					(* Valuto la posizione attuale Y e la posizione di destinazione Y e l'ingombro massimo che posso avere durante il transito *)
					IF (Mission^.YPick - IngombroOttimizzatoY_InTransito/2 - OffsetSicurezza_Y <= WorkFootprint^[5].Y) OR //Posizione Pinza - Metà ingombro - Offset sicurezza <= Ingombro colonna 
						(Mission^.YPick + IngombroOttimizzatoY_InTransito/2 + OffsetSicurezza_Y >= WorkFootprint^[6].Y) THEN //Posizione Pinza - Metà ingombro - Offset sicurezza <= Ingombro colonna 
							Pinza_InIngombroColonne_Transito := TRUE;
					ELSE
							Pinza_InIngombroColonne_Transito := FALSE;
					END_IF
			END_CASE		
			(* Se sono in ingombro nella posizione attuale o nella posizione di destinazione, devo andare fuori-ingombro con la Y *)
			IF (Pinza_InIngombroColonne_Attuale OR Pinza_InIngombroColonne_Destinazione OR Pinza_InIngombroColonne_Transito) AND AreaInLavoroPositivaNegativa THEN 
				IF (AsseXInFinestraDiRiposo AND AsseYInFinestraDiRiposo AND AsseJInFinestraDiRiposo) THEN //Se sono in finestra di riposo con tutti gli assi non devo andare fuori-ingombro con la Y
					FuoriIngombroYNecessarioTMP := FALSE;
				ELSE
					FuoriIngombroYNecessarioTMP := TRUE;
				END_IF
			ELSE
				FuoriIngombroYNecessarioTMP := FALSE;
			END_IF
		END_IF
				
	WAMANAGER_CICLO_PRELIEVO_FALDA_VUOTI_END:
		CalcolaIngombro := TRUE;	
		
	WAMANAGER_CICLO_DEPOSITO_FALDA_VUOTI_RUN:
		IF CalcolaIngombro THEN
			CalcolaIngombro := FALSE;
			(* Definisco il tipo di area in cui si trova a lavorare il pallettizzatore *)
			AreaInLavoroPositiva := FALSE;
			AreaInLavoroNegativa := FALSE;
			AreaInLavoroPositivaNegativa := FALSE; 
			IF ModuleAx_X^.Ax^.AxRef^.NcToPlc.ActPos >= (WorkFootprint^[5].X + WorkFootprint^[5].XDim) AND 	//se la piazzola di prelievo ha quota maggiore rispetto le colonne centrali
				WorkArea^[Mission^.PPlace].X >= (WorkFootprint^[5].X + WorkFootprint^[5].XDim)  THEN //la piazzola di deposito è nella campata positiva
					AreaInLavoroPositiva := TRUE;
			ELSIF ModuleAx_X^.Ax^.AxRef^.NcToPlc.ActPos <= WorkFootprint^[5].X AND 	//se la piazzola di prelievo ha quota maggiore della piazzola di deposito e
				WorkArea^[Mission^.PPlace].X <= WorkFootprint^[5].X  THEN //la piazzola di deposito è nella campata negativa
					AreaInLavoroNegativa := TRUE;
			ELSE
				AreaInLavoroPositiva := FALSE;
				AreaInLavoroNegativa := FALSE;
				AreaInLavoroPositivaNegativa := TRUE;
			END_IF
			
			(**************************************************************************************************************************************************)
			(* Ingombro ottimizzato della pinza sul punto di prelievo *)
			(**************************************************************************************************************************************************)
			IngombroOttimizzatoX_InPuntoDiPrelievo := ABS(IngombroSuperficialePinzaMAX * SIN(deg_to_rad((ATAN(Larghezza/Lunghezza)*1/0.017+ Mission^.JPick))));
			IngombroOttimizzatoY_InPuntoDiPrelievo := ABS(IngombroSuperficialePinzaMAX * COS(deg_to_rad((ATAN(Larghezza/Lunghezza)*1/0.017+ Mission^.JPick))));
			(**************************************************************************************************************************************************)
			(* Ingombro ottimizzato della pinza sul punto di deposito *)
			(**************************************************************************************************************************************************)
			IngombroOttimizzatoX_InPuntoDiDeposito := ABS(IngombroSuperficialePinzaMAX * SIN(deg_to_rad((ATAN(Larghezza/Lunghezza)*1/0.017+ Mission^.JPlace))));
			IngombroOttimizzatoY_InPuntoDiDeposito := ABS(IngombroSuperficialePinzaMAX * COS(deg_to_rad((ATAN(Larghezza/Lunghezza)*1/0.017+ Mission^.JPlace))));
						
			(**************************************************************************************************************************************************)
			(**************************************************************************************************************************************************)
						
			(* Valuto la direzione della X *)
			DirezioneXPositiva := TFDirezioneAssePositiva(Posizione_Attuale:=ModuleAX_X^.Ax^.Status.ActPosition,Posizione_Finale:=Mission^.XPick);
			DirezioneXNegativa := NOT DirezioneXPositiva;
				
			(* Valuto se gli assi sono in finestra di prelievo *)
			AsseXInFinestraDiRiposo := TFAsseInFinestra(Posizione_Attuale:=ModuleAx_X^.Ax^.AxRef^.NcToPlc.ActPos,Posizione_Finale:=Mission^.XPick,FinestraDiControllo:=10);
			AsseYInFinestraDiRiposo := TFAsseInFinestra(Posizione_Attuale:=ModuleAx_Y^.Ax^.AxRef^.NcToPlc.ActPos,Posizione_Finale:=Mission^.YPick,FinestraDiControllo:=10);
			AsseJInFinestraDiRiposo := TFAsseInFinestra(Posizione_Attuale:=ModuleAx_J^.Ax^.AxRef^.NcToPlc.ActPos,Posizione_Finale:=Mission^.JPick,FinestraDiControllo:=5);
			(* Valuto se gli assi sono in finestra di destinazione *)
			AsseXInFinestraDiDestinazione := TFAsseInFinestra(Posizione_Attuale:=ModuleAx_X^.Ax^.AxRef^.NcToPlc.ActPos,Posizione_Finale:=Mission^.XPick,FinestraDiControllo:=10);
			AsseYInFinestraDiDestinazione := TFAsseInFinestra(Posizione_Attuale:=ModuleAx_Y^.Ax^.AxRef^.NcToPlc.ActPos,Posizione_Finale:=Mission^.YPick,FinestraDiControllo:=10);
			AsseJInFinestraDiDestinazione := TFAsseInFinestra(Posizione_Attuale:=ModuleAx_J^.Ax^.AxRef^.NcToPlc.ActPos,Posizione_Finale:=Mission^.JPick,FinestraDiControllo:=5);
			
			(**************************************************************************************************************************************************)
			(* Ingombro MASSIMO della pinza durante il transito *)
			(**************************************************************************************************************************************************)
			//Calcolo ingombro attuale
			IngombroOttimizzatoX_InTransito := ABS(IngombroSuperficialePinzaMAX * SIN(deg_to_rad((ATAN(Larghezza/Lunghezza)*1/0.017+ ModuleAx_J^.Ax^.AxRef^.NcToPlc.ActPos)))); //Ingombro Attuale direzione X
			IngombroOttimizzatoY_InTransito := ABS(IngombroSuperficialePinzaMAX * COS(deg_to_rad((ATAN(Larghezza/Lunghezza)*1/0.017+ ModuleAx_J^.Ax^.AxRef^.NcToPlc.ActPos)))); //Ingombro Attuale direzione Y		
			IF NOT AsseJInFinestraDiDestinazione THEN
				IF REAL_TO_INT(ModuleAx_J^.Ax^.AxRef^.NcToPlc.ActPos) <= REAL_TO_INT(Mission^.JPick) THEN
					FOR Angolo := REAL_TO_INT(ModuleAx_J^.Ax^.AxRef^.NcToPlc.ActPos) TO REAL_TO_INT(Mission^.JPick)  DO
						IF IngombroOttimizzatoX_InTransito < ABS(IngombroSuperficialePinzaMAX * SIN(deg_to_rad((ATAN(Larghezza/Lunghezza)*1/0.017+ Angolo)))) THEN
							IngombroOttimizzatoX_InTransito := ABS(IngombroSuperficialePinzaMAX * SIN(deg_to_rad((ATAN(Larghezza/Lunghezza)*1/0.017+ Angolo)))) ;
						END_IF
						IF IngombroOttimizzatoY_InTransito < ABS(IngombroSuperficialePinzaMAX * COS(deg_to_rad((ATAN(Larghezza/Lunghezza)*1/0.017+ Angolo)))) THEN
							IngombroOttimizzatoY_InTransito := ABS(IngombroSuperficialePinzaMAX * COS(deg_to_rad((ATAN(Larghezza/Lunghezza)*1/0.017+ Angolo))));
						END_IF
					END_FOR
				END_IF
			END_IF
		
			(* Valutazione colonne in base al verso del pallettizzatore *)
			CASE VERSO_PALLETTIZZATORE OF
				PALLETTIZZATORE_DX:	// Colonna 6:DX, 5:SX
					(* Valuto la posizione attuale *)
					IF (ModuleAX_Y^.Ax^.Status.ActPosition - IngombroY/2 - OffsetSicurezza_Y <= WorkFootprint^[6].Y) OR //Posizione Pinza - Metà ingombro - Offset sicurezza <= Ingombro colonna 
						(ModuleAX_Y^.Ax^.Status.ActPosition + IngombroY/2 + OffsetSicurezza_Y >= WorkFootprint^[5].Y) THEN //Posizione Pinza - Metà ingombro - Offset sicurezza <= Ingombro colonna 
							Pinza_InIngombroColonne_Attuale := TRUE;
					ELSE
							Pinza_InIngombroColonne_Attuale := FALSE;
					END_IF
					(* Valuto la posizione futura - Missione di prelievo *)
					IF (Mission^.YPick - IngombroOttimizzatoX_InPuntoDiPrelievo/2 - OffsetSicurezza_Y <= WorkFootprint^[6].Y) OR //Posizione Pinza - Metà ingombro - Offset sicurezza <= Ingombro colonna 
						(Mission^.YPick + IngombroOttimizzatoX_InPuntoDiPrelievo/2 + OffsetSicurezza_Y >= WorkFootprint^[5].Y) THEN //Posizione Pinza - Metà ingombro - Offset sicurezza <= Ingombro colonna 
							Pinza_InIngombroColonne_Destinazione := TRUE;
					ELSE
							Pinza_InIngombroColonne_Destinazione := FALSE;
					END_IF
					
					(* Valuto la posizione futura - Missione di Deposito *)
					IF (Mission^.YPick - IngombroOttimizzatoX_InPuntoDiDeposito/2 - OffsetSicurezza_Y <= WorkFootprint^[6].Y) OR //Posizione Pinza - Metà ingombro - Offset sicurezza <= Ingombro colonna 
						(Mission^.YPick + IngombroOttimizzatoX_InPuntoDiDeposito/2 + OffsetSicurezza_Y >= WorkFootprint^[5].Y) THEN //Posizione Pinza - Metà ingombro - Offset sicurezza <= Ingombro colonna 
							Pinza_InIngombroColonne_Destinazione := TRUE;
					ELSE
							Pinza_InIngombroColonne_Destinazione := FALSE;
					END_IF
					
					(* Valuto la posizione attuale Y e la posizione di destinazione Y e l'ingombro massimo che posso avere durante il transito *)
					IF (Mission^.YPick - IngombroOttimizzatoY_InTransito/2 - OffsetSicurezza_Y <= WorkFootprint^[6].Y) OR //Posizione Pinza - Metà ingombro - Offset sicurezza <= Ingombro colonna 
						(Mission^.YPick + IngombroOttimizzatoY_InTransito/2 + OffsetSicurezza_Y >= WorkFootprint^[5].Y) THEN //Posizione Pinza - Metà ingombro - Offset sicurezza <= Ingombro colonna 
							Pinza_InIngombroColonne_Transito := TRUE;
					ELSE
							Pinza_InIngombroColonne_Transito := FALSE;
					END_IF
						
				PALLETTIZZATORE_SX: // Colonna 6:SX, 5:DX
					(* Valuto la posizione attuale *)
					IF (ModuleAX_Y^.Ax^.Status.ActPosition - IngombroY/2 - OffsetSicurezza_Y <= WorkFootprint^[5].Y) OR //Posizione Pinza - Metà ingombro - Offset sicurezza <= Ingombro colonna 
						(ModuleAX_Y^.Ax^.Status.ActPosition + IngombroY/2 + OffsetSicurezza_Y >= WorkFootprint^[6].Y) THEN //Posizione Pinza - Metà ingombro - Offset sicurezza <= Ingombro colonna 
							Pinza_InIngombroColonne_Attuale := TRUE;
					ELSE
							Pinza_InIngombroColonne_Attuale := FALSE;
					END_IF
					(* Valuto la posizione futura - Missione di prelievo *)
					IF (Mission^.YPick - IngombroOttimizzatoX_InPuntoDiPrelievo/2 - OffsetSicurezza_Y <= WorkFootprint^[5].Y) OR //Posizione Pinza - Metà ingombro - Offset sicurezza <= Ingombro colonna 
						(Mission^.YPick + IngombroOttimizzatoX_InPuntoDiPrelievo/2 + OffsetSicurezza_Y >= WorkFootprint^[6].Y) THEN //Posizione Pinza - Metà ingombro - Offset sicurezza <= Ingombro colonna 
							Pinza_InIngombroColonne_Destinazione := TRUE;
					ELSE
							Pinza_InIngombroColonne_Destinazione := FALSE;
					END_IF
					
					(* Valuto la posizione futura - Missione di Deposito *)
					IF (Mission^.YPick - IngombroOttimizzatoX_InPuntoDiDeposito/2 - OffsetSicurezza_Y <= WorkFootprint^[5].Y) OR //Posizione Pinza - Metà ingombro - Offset sicurezza <= Ingombro colonna 
						(Mission^.YPick + IngombroOttimizzatoX_InPuntoDiDeposito/2 + OffsetSicurezza_Y >= WorkFootprint^[6].Y) THEN //Posizione Pinza - Metà ingombro - Offset sicurezza <= Ingombro colonna 
							Pinza_InIngombroColonne_Destinazione := TRUE;
					ELSE
							Pinza_InIngombroColonne_Destinazione := FALSE;
					END_IF
					
					(* Valuto la posizione attuale Y e la posizione di destinazione Y e l'ingombro massimo che posso avere durante il transito *)
					IF (Mission^.YPick - IngombroOttimizzatoY_InTransito/2 - OffsetSicurezza_Y <= WorkFootprint^[5].Y) OR //Posizione Pinza - Metà ingombro - Offset sicurezza <= Ingombro colonna 
						(Mission^.YPick + IngombroOttimizzatoY_InTransito/2 + OffsetSicurezza_Y >= WorkFootprint^[6].Y) THEN //Posizione Pinza - Metà ingombro - Offset sicurezza <= Ingombro colonna 
							Pinza_InIngombroColonne_Transito := TRUE;
					ELSE
							Pinza_InIngombroColonne_Transito := FALSE;
					END_IF
			END_CASE		
			(* Se sono in ingombro nella posizione attuale o nella posizione di destinazione, devo andare fuori-ingombro con la Y *)
			IF (Pinza_InIngombroColonne_Attuale OR Pinza_InIngombroColonne_Destinazione OR Pinza_InIngombroColonne_Transito) AND AreaInLavoroPositivaNegativa THEN 
				IF (AsseXInFinestraDiRiposo AND AsseYInFinestraDiRiposo AND AsseJInFinestraDiRiposo) THEN //Se sono in finestra di riposo con tutti gli assi non devo andare fuori-ingombro con la Y
					FuoriIngombroYNecessarioTMP := FALSE;
				ELSE
					FuoriIngombroYNecessarioTMP := TRUE;
				END_IF
			ELSE
				FuoriIngombroYNecessarioTMP := FALSE;
			END_IF
		END_IF
								
	WAMANAGER_CICLO_DEPOSITO_FALDA_VUOTI_END:
		CalcolaIngombro := TRUE;	
	
	WAMANAGER_CICLO_FALDA_INIT:
		CalcolaIngombro := TRUE;	
	
	WAMANAGER_CICLO_PRELIEVO_FALDA_RUN:
		IF CalcolaIngombro THEN
			CalcolaIngombro := FALSE;
			(* Definisco il tipo di area in cui si trova a lavorare il pallettizzatore *)
			AreaInLavoroPositiva := FALSE;
			AreaInLavoroNegativa := FALSE;
			AreaInLavoroPositivaNegativa := TRUE; 
			
			(**************************************************************************************************************************************************)
			(* Ingombro ottimizzato della pinza sul punto di prelievo *)
			(**************************************************************************************************************************************************)
			IngombroOttimizzatoX_InPuntoDiPrelievo := ABS(IngombroSuperficialePinzaMAX * SIN(deg_to_rad((ATAN(Larghezza/Lunghezza)*1/0.017+ Mission^.JPick))));
			IngombroOttimizzatoY_InPuntoDiPrelievo := ABS(IngombroSuperficialePinzaMAX * COS(deg_to_rad((ATAN(Larghezza/Lunghezza)*1/0.017+ Mission^.JPick))));
			(**************************************************************************************************************************************************)
			(* Ingombro ottimizzato della pinza sul punto di deposito *)
			(**************************************************************************************************************************************************)
			IngombroOttimizzatoX_InPuntoDiDeposito := ABS(IngombroSuperficialePinzaMAX * SIN(deg_to_rad((ATAN(Larghezza/Lunghezza)*1/0.017+ Mission^.JPlace))));
			IngombroOttimizzatoY_InPuntoDiDeposito := ABS(IngombroSuperficialePinzaMAX * COS(deg_to_rad((ATAN(Larghezza/Lunghezza)*1/0.017+ Mission^.JPlace))));
						
			(**************************************************************************************************************************************************)
			(**************************************************************************************************************************************************)
						
			(* Valuto la direzione della X *)
			DirezioneXPositiva := TFDirezioneAssePositiva(Posizione_Attuale:=ModuleAX_X^.Ax^.Status.ActPosition,Posizione_Finale:=Mission^.XPick);
			DirezioneXNegativa := NOT DirezioneXPositiva;
				
			(* Valuto se gli assi sono in finestra di prelievo *)
			AsseXInFinestraDiRiposo := TFAsseInFinestra(Posizione_Attuale:=ModuleAx_X^.Ax^.AxRef^.NcToPlc.ActPos,Posizione_Finale:=Mission^.XPick,FinestraDiControllo:=10);
			AsseYInFinestraDiRiposo := TFAsseInFinestra(Posizione_Attuale:=ModuleAx_Y^.Ax^.AxRef^.NcToPlc.ActPos,Posizione_Finale:=Mission^.YPick,FinestraDiControllo:=10);
			AsseJInFinestraDiRiposo := TFAsseInFinestra(Posizione_Attuale:=ModuleAx_J^.Ax^.AxRef^.NcToPlc.ActPos,Posizione_Finale:=Mission^.JPick,FinestraDiControllo:=5);
			(* Valuto se gli assi sono in finestra di destinazione *)
			AsseXInFinestraDiDestinazione := TFAsseInFinestra(Posizione_Attuale:=ModuleAx_X^.Ax^.AxRef^.NcToPlc.ActPos,Posizione_Finale:=Mission^.XPick,FinestraDiControllo:=10);
			AsseYInFinestraDiDestinazione := TFAsseInFinestra(Posizione_Attuale:=ModuleAx_Y^.Ax^.AxRef^.NcToPlc.ActPos,Posizione_Finale:=Mission^.YPick,FinestraDiControllo:=10);
			AsseJInFinestraDiDestinazione := TFAsseInFinestra(Posizione_Attuale:=ModuleAx_J^.Ax^.AxRef^.NcToPlc.ActPos,Posizione_Finale:=Mission^.JPick,FinestraDiControllo:=5);
			
			(**************************************************************************************************************************************************)
			(* Ingombro MASSIMO della pinza durante il transito *)
			(**************************************************************************************************************************************************)
			//Calcolo ingombro attuale
			IngombroOttimizzatoX_InTransito := ABS(IngombroSuperficialePinzaMAX * SIN(deg_to_rad((ATAN(Larghezza/Lunghezza)*1/0.017+ ModuleAx_J^.Ax^.AxRef^.NcToPlc.ActPos)))); //Ingombro Attuale direzione X
			IngombroOttimizzatoY_InTransito := ABS(IngombroSuperficialePinzaMAX * COS(deg_to_rad((ATAN(Larghezza/Lunghezza)*1/0.017+ ModuleAx_J^.Ax^.AxRef^.NcToPlc.ActPos)))); //Ingombro Attuale direzione Y		
			IF NOT AsseJInFinestraDiDestinazione THEN
				IF REAL_TO_INT(ModuleAx_J^.Ax^.AxRef^.NcToPlc.ActPos) <= REAL_TO_INT(Mission^.JPick) THEN
					FOR Angolo := REAL_TO_INT(ModuleAx_J^.Ax^.AxRef^.NcToPlc.ActPos) TO REAL_TO_INT(Mission^.JPick)  DO
						IF IngombroOttimizzatoX_InTransito < ABS(IngombroSuperficialePinzaMAX * SIN(deg_to_rad((ATAN(Larghezza/Lunghezza)*1/0.017+ Angolo)))) THEN
							IngombroOttimizzatoX_InTransito := ABS(IngombroSuperficialePinzaMAX * SIN(deg_to_rad((ATAN(Larghezza/Lunghezza)*1/0.017+ Angolo)))) ;
						END_IF
						IF IngombroOttimizzatoY_InTransito < ABS(IngombroSuperficialePinzaMAX * COS(deg_to_rad((ATAN(Larghezza/Lunghezza)*1/0.017+ Angolo)))) THEN
							IngombroOttimizzatoY_InTransito := ABS(IngombroSuperficialePinzaMAX * COS(deg_to_rad((ATAN(Larghezza/Lunghezza)*1/0.017+ Angolo))));
						END_IF
					END_FOR
				END_IF
			END_IF
		
			(* Valutazione colonne in base al verso del pallettizzatore *)
			CASE VERSO_PALLETTIZZATORE OF
				PALLETTIZZATORE_DX:	// Colonna 6:DX, 5:SX
					(* Valuto la posizione attuale *)
					IF (ModuleAX_Y^.Ax^.Status.ActPosition - IngombroY/2 - OffsetSicurezza_Y <= WorkFootprint^[6].Y) OR //Posizione Pinza - Metà ingombro - Offset sicurezza <= Ingombro colonna 
						(ModuleAX_Y^.Ax^.Status.ActPosition + IngombroY/2 + OffsetSicurezza_Y >= WorkFootprint^[5].Y) THEN //Posizione Pinza - Metà ingombro - Offset sicurezza <= Ingombro colonna 
							Pinza_InIngombroColonne_Attuale := TRUE;
					ELSE
							Pinza_InIngombroColonne_Attuale := FALSE;
					END_IF
					(* Valuto la posizione futura - Missione di prelievo *)
					IF (Mission^.YPick - IngombroOttimizzatoX_InPuntoDiPrelievo/2 - OffsetSicurezza_Y <= WorkFootprint^[6].Y) OR //Posizione Pinza - Metà ingombro - Offset sicurezza <= Ingombro colonna 
						(Mission^.YPick + IngombroOttimizzatoX_InPuntoDiPrelievo/2 + OffsetSicurezza_Y >= WorkFootprint^[5].Y) THEN //Posizione Pinza - Metà ingombro - Offset sicurezza <= Ingombro colonna 
							Pinza_InIngombroColonne_Destinazione := TRUE;
					ELSE
							Pinza_InIngombroColonne_Destinazione := FALSE;
					END_IF
					
					(* Valuto la posizione futura - Missione di Deposito *)
					IF (Mission^.YPick - IngombroOttimizzatoX_InPuntoDiDeposito/2 - OffsetSicurezza_Y <= WorkFootprint^[6].Y) OR //Posizione Pinza - Metà ingombro - Offset sicurezza <= Ingombro colonna 
						(Mission^.YPick + IngombroOttimizzatoX_InPuntoDiDeposito/2 + OffsetSicurezza_Y >= WorkFootprint^[5].Y) THEN //Posizione Pinza - Metà ingombro - Offset sicurezza <= Ingombro colonna 
							Pinza_InIngombroColonne_Destinazione := TRUE;
					ELSE
							Pinza_InIngombroColonne_Destinazione := FALSE;
					END_IF
					
					(* Valuto la posizione attuale Y e la posizione di destinazione Y e l'ingombro massimo che posso avere durante il transito *)
					IF (Mission^.YPick - IngombroOttimizzatoY_InTransito/2 - OffsetSicurezza_Y <= WorkFootprint^[6].Y) OR //Posizione Pinza - Metà ingombro - Offset sicurezza <= Ingombro colonna 
						(Mission^.YPick + IngombroOttimizzatoY_InTransito/2 + OffsetSicurezza_Y >= WorkFootprint^[5].Y) THEN //Posizione Pinza - Metà ingombro - Offset sicurezza <= Ingombro colonna 
							Pinza_InIngombroColonne_Transito := TRUE;
					ELSE
							Pinza_InIngombroColonne_Transito := FALSE;
					END_IF
						
				PALLETTIZZATORE_SX: // Colonna 6:SX, 5:DX
					(* Valuto la posizione attuale *)
					IF (ModuleAX_Y^.Ax^.Status.ActPosition - IngombroY/2 - OffsetSicurezza_Y <= WorkFootprint^[5].Y) OR //Posizione Pinza - Metà ingombro - Offset sicurezza <= Ingombro colonna 
						(ModuleAX_Y^.Ax^.Status.ActPosition + IngombroY/2 + OffsetSicurezza_Y >= WorkFootprint^[6].Y) THEN //Posizione Pinza - Metà ingombro - Offset sicurezza <= Ingombro colonna 
							Pinza_InIngombroColonne_Attuale := TRUE;
					ELSE
							Pinza_InIngombroColonne_Attuale := FALSE;
					END_IF
					(* Valuto la posizione futura - Missione di prelievo *)
					IF (Mission^.YPick - IngombroOttimizzatoX_InPuntoDiPrelievo/2 - OffsetSicurezza_Y <= WorkFootprint^[5].Y) OR //Posizione Pinza - Metà ingombro - Offset sicurezza <= Ingombro colonna 
						(Mission^.YPick + IngombroOttimizzatoX_InPuntoDiPrelievo/2 + OffsetSicurezza_Y >= WorkFootprint^[6].Y) THEN //Posizione Pinza - Metà ingombro - Offset sicurezza <= Ingombro colonna 
							Pinza_InIngombroColonne_Destinazione := TRUE;
					ELSE
							Pinza_InIngombroColonne_Destinazione := FALSE;
					END_IF
					
					(* Valuto la posizione futura - Missione di Deposito *)
					IF (Mission^.YPick - IngombroOttimizzatoX_InPuntoDiDeposito/2 - OffsetSicurezza_Y <= WorkFootprint^[5].Y) OR //Posizione Pinza - Metà ingombro - Offset sicurezza <= Ingombro colonna 
						(Mission^.YPick + IngombroOttimizzatoX_InPuntoDiDeposito/2 + OffsetSicurezza_Y >= WorkFootprint^[6].Y) THEN //Posizione Pinza - Metà ingombro - Offset sicurezza <= Ingombro colonna 
							Pinza_InIngombroColonne_Destinazione := TRUE;
					ELSE
							Pinza_InIngombroColonne_Destinazione := FALSE;
					END_IF
					
					(* Valuto la posizione attuale Y e la posizione di destinazione Y e l'ingombro massimo che posso avere durante il transito *)
					IF (Mission^.YPick - IngombroOttimizzatoY_InTransito/2 - OffsetSicurezza_Y <= WorkFootprint^[5].Y) OR //Posizione Pinza - Metà ingombro - Offset sicurezza <= Ingombro colonna 
						(Mission^.YPick + IngombroOttimizzatoY_InTransito/2 + OffsetSicurezza_Y >= WorkFootprint^[6].Y) THEN //Posizione Pinza - Metà ingombro - Offset sicurezza <= Ingombro colonna 
							Pinza_InIngombroColonne_Transito := TRUE;
					ELSE
							Pinza_InIngombroColonne_Transito := FALSE;
					END_IF
			END_CASE		
			(* Se sono in ingombro nella posizione attuale o nella posizione di destinazione, devo andare fuori-ingombro con la Y *)
			IF (Pinza_InIngombroColonne_Attuale OR Pinza_InIngombroColonne_Destinazione OR Pinza_InIngombroColonne_Transito) THEN 
				IF (AsseXInFinestraDiRiposo AND AsseYInFinestraDiRiposo AND AsseJInFinestraDiRiposo) THEN //Se sono in finestra di riposo con tutti gli assi non devo andare fuori-ingombro con la Y
					FuoriIngombroYNecessarioTMP := FALSE;
				ELSE
					FuoriIngombroYNecessarioTMP := TRUE;
				END_IF
			ELSE
				FuoriIngombroYNecessarioTMP := FALSE;
			END_IF
		END_IF		
																
	WAMANAGER_CICLO_PRELIEVO_FALDA_END:
		CalcolaIngombro := TRUE;	
			
	WAMANAGER_CICLO_DEPOSITO_FALDA_RUN:
		IF CalcolaIngombro THEN
			CalcolaIngombro := FALSE;
			(* Definisco il tipo di area in cui si trova a lavorare il pallettizzatore *)
			AreaInLavoroPositiva := FALSE;
			AreaInLavoroNegativa := FALSE;
			AreaInLavoroPositivaNegativa := TRUE; 
			
			IF ModuleAx_X^.Ax^.AxRef^.NcToPlc.ActPos >= (WorkFootprint^[5].X + WorkFootprint^[5].XDim) AND 	//se la piazzola di prelievo ha quota maggiore rispetto le colonne centrali
				WorkArea^[Mission^.PPlace].X >= (WorkFootprint^[5].X + WorkFootprint^[5].XDim)  THEN //la piazzola di deposito è nella campata positiva
					AreaInLavoroPositiva := TRUE;
			ELSIF ModuleAx_X^.Ax^.AxRef^.NcToPlc.ActPos <= WorkFootprint^[5].X AND 	//se la piazzola di prelievo ha quota maggiore della piazzola di deposito e
				WorkArea^[Mission^.PPlace].X <= WorkFootprint^[5].X  THEN //la piazzola di deposito è nella campata negativa
					AreaInLavoroNegativa := TRUE;
			ELSE
				AreaInLavoroPositiva := FALSE;
				AreaInLavoroNegativa := FALSE;
				AreaInLavoroPositivaNegativa := TRUE;
			END_IF
			
			(**************************************************************************************************************************************************)
			(* Ingombro ottimizzato della pinza sul punto di prelievo *)
			(**************************************************************************************************************************************************)
			IngombroOttimizzatoX_InPuntoDiPrelievo := ABS(IngombroSuperficialePinzaMAX * SIN(deg_to_rad((ATAN(Larghezza/Lunghezza)*1/0.017+ Mission^.JPick))));
			IngombroOttimizzatoY_InPuntoDiPrelievo := ABS(IngombroSuperficialePinzaMAX * COS(deg_to_rad((ATAN(Larghezza/Lunghezza)*1/0.017+ Mission^.JPick))));
			(**************************************************************************************************************************************************)
			(* Ingombro ottimizzato della pinza sul punto di deposito *)
			(**************************************************************************************************************************************************)
			IngombroOttimizzatoX_InPuntoDiDeposito := ABS(IngombroSuperficialePinzaMAX * SIN(deg_to_rad((ATAN(Larghezza/Lunghezza)*1/0.017+ Mission^.JPlace))));
			IngombroOttimizzatoY_InPuntoDiDeposito := ABS(IngombroSuperficialePinzaMAX * COS(deg_to_rad((ATAN(Larghezza/Lunghezza)*1/0.017+ Mission^.JPlace))));
						
			(**************************************************************************************************************************************************)
			(**************************************************************************************************************************************************)
						
			(* Valuto la direzione della X *)
			DirezioneXPositiva := TFDirezioneAssePositiva(Posizione_Attuale:=ModuleAX_X^.Ax^.Status.ActPosition,Posizione_Finale:=Mission^.XPick);
			DirezioneXNegativa := NOT DirezioneXPositiva;
				
			(* Valuto se gli assi sono in finestra di prelievo *)
			AsseXInFinestraDiRiposo := TFAsseInFinestra(Posizione_Attuale:=ModuleAx_X^.Ax^.AxRef^.NcToPlc.ActPos,Posizione_Finale:=Mission^.XPick,FinestraDiControllo:=10);
			AsseYInFinestraDiRiposo := TFAsseInFinestra(Posizione_Attuale:=ModuleAx_Y^.Ax^.AxRef^.NcToPlc.ActPos,Posizione_Finale:=Mission^.YPick,FinestraDiControllo:=10);
			AsseJInFinestraDiRiposo := TFAsseInFinestra(Posizione_Attuale:=ModuleAx_J^.Ax^.AxRef^.NcToPlc.ActPos,Posizione_Finale:=Mission^.JPick,FinestraDiControllo:=5);
			(* Valuto se gli assi sono in finestra di destinazione *)
			AsseXInFinestraDiDestinazione := TFAsseInFinestra(Posizione_Attuale:=ModuleAx_X^.Ax^.AxRef^.NcToPlc.ActPos,Posizione_Finale:=Mission^.XPick,FinestraDiControllo:=10);
			AsseYInFinestraDiDestinazione := TFAsseInFinestra(Posizione_Attuale:=ModuleAx_Y^.Ax^.AxRef^.NcToPlc.ActPos,Posizione_Finale:=Mission^.YPick,FinestraDiControllo:=10);
			AsseJInFinestraDiDestinazione := TFAsseInFinestra(Posizione_Attuale:=ModuleAx_J^.Ax^.AxRef^.NcToPlc.ActPos,Posizione_Finale:=Mission^.JPick,FinestraDiControllo:=5);
			
			(**************************************************************************************************************************************************)
			(* Ingombro MASSIMO della pinza durante il transito *)
			(**************************************************************************************************************************************************)
			//Calcolo ingombro attuale
			IngombroOttimizzatoX_InTransito := ABS(IngombroSuperficialePinzaMAX * SIN(deg_to_rad((ATAN(Larghezza/Lunghezza)*1/0.017+ ModuleAx_J^.Ax^.AxRef^.NcToPlc.ActPos)))); //Ingombro Attuale direzione X
			IngombroOttimizzatoY_InTransito := ABS(IngombroSuperficialePinzaMAX * COS(deg_to_rad((ATAN(Larghezza/Lunghezza)*1/0.017+ ModuleAx_J^.Ax^.AxRef^.NcToPlc.ActPos)))); //Ingombro Attuale direzione Y		
			IF NOT AsseJInFinestraDiDestinazione THEN
				IF REAL_TO_INT(ModuleAx_J^.Ax^.AxRef^.NcToPlc.ActPos) <= REAL_TO_INT(Mission^.JPick) THEN
					FOR Angolo := REAL_TO_INT(ModuleAx_J^.Ax^.AxRef^.NcToPlc.ActPos) TO REAL_TO_INT(Mission^.JPick)  DO
						IF IngombroOttimizzatoX_InTransito < ABS(IngombroSuperficialePinzaMAX * SIN(deg_to_rad((ATAN(Larghezza/Lunghezza)*1/0.017+ Angolo)))) THEN
							IngombroOttimizzatoX_InTransito := ABS(IngombroSuperficialePinzaMAX * SIN(deg_to_rad((ATAN(Larghezza/Lunghezza)*1/0.017+ Angolo)))) ;
						END_IF
						IF IngombroOttimizzatoY_InTransito < ABS(IngombroSuperficialePinzaMAX * COS(deg_to_rad((ATAN(Larghezza/Lunghezza)*1/0.017+ Angolo)))) THEN
							IngombroOttimizzatoY_InTransito := ABS(IngombroSuperficialePinzaMAX * COS(deg_to_rad((ATAN(Larghezza/Lunghezza)*1/0.017+ Angolo))));
						END_IF
					END_FOR
				END_IF
			END_IF
		
			(* Valutazione colonne in base al verso del pallettizzatore *)
			CASE VERSO_PALLETTIZZATORE OF
				PALLETTIZZATORE_DX:	// Colonna 6:DX, 5:SX
					(* Valuto la posizione attuale *)
					IF (ModuleAX_Y^.Ax^.Status.ActPosition - IngombroY/2 - OffsetSicurezza_Y <= WorkFootprint^[6].Y) OR //Posizione Pinza - Metà ingombro - Offset sicurezza <= Ingombro colonna 
						(ModuleAX_Y^.Ax^.Status.ActPosition + IngombroY/2 + OffsetSicurezza_Y >= WorkFootprint^[5].Y) THEN //Posizione Pinza - Metà ingombro - Offset sicurezza <= Ingombro colonna 
							Pinza_InIngombroColonne_Attuale := TRUE;
					ELSE
							Pinza_InIngombroColonne_Attuale := FALSE;
					END_IF
					(* Valuto la posizione futura - Missione di prelievo *)
					IF (Mission^.YPick - IngombroOttimizzatoX_InPuntoDiPrelievo/2 - OffsetSicurezza_Y <= WorkFootprint^[6].Y) OR //Posizione Pinza - Metà ingombro - Offset sicurezza <= Ingombro colonna 
						(Mission^.YPick + IngombroOttimizzatoX_InPuntoDiPrelievo/2 + OffsetSicurezza_Y >= WorkFootprint^[5].Y) THEN //Posizione Pinza - Metà ingombro - Offset sicurezza <= Ingombro colonna 
							Pinza_InIngombroColonne_Destinazione := TRUE;
					ELSE
							Pinza_InIngombroColonne_Destinazione := FALSE;
					END_IF
					
					(* Valuto la posizione futura - Missione di Deposito *)
					IF (Mission^.YPick - IngombroOttimizzatoX_InPuntoDiDeposito/2 - OffsetSicurezza_Y <= WorkFootprint^[6].Y) OR //Posizione Pinza - Metà ingombro - Offset sicurezza <= Ingombro colonna 
						(Mission^.YPick + IngombroOttimizzatoX_InPuntoDiDeposito/2 + OffsetSicurezza_Y >= WorkFootprint^[5].Y) THEN //Posizione Pinza - Metà ingombro - Offset sicurezza <= Ingombro colonna 
							Pinza_InIngombroColonne_Destinazione := TRUE;
					ELSE
							Pinza_InIngombroColonne_Destinazione := FALSE;
					END_IF
					
					(* Valuto la posizione attuale Y e la posizione di destinazione Y e l'ingombro massimo che posso avere durante il transito *)
					IF (Mission^.YPick - IngombroOttimizzatoY_InTransito/2 - OffsetSicurezza_Y <= WorkFootprint^[6].Y) OR //Posizione Pinza - Metà ingombro - Offset sicurezza <= Ingombro colonna 
						(Mission^.YPick + IngombroOttimizzatoY_InTransito/2 + OffsetSicurezza_Y >= WorkFootprint^[5].Y) THEN //Posizione Pinza - Metà ingombro - Offset sicurezza <= Ingombro colonna 
							Pinza_InIngombroColonne_Transito := TRUE;
					ELSE
							Pinza_InIngombroColonne_Transito := FALSE;
					END_IF
						
				PALLETTIZZATORE_SX: // Colonna 6:SX, 5:DX
					(* Valuto la posizione attuale *)
					IF (ModuleAX_Y^.Ax^.Status.ActPosition - IngombroY/2 - OffsetSicurezza_Y <= WorkFootprint^[5].Y) OR //Posizione Pinza - Metà ingombro - Offset sicurezza <= Ingombro colonna 
						(ModuleAX_Y^.Ax^.Status.ActPosition + IngombroY/2 + OffsetSicurezza_Y >= WorkFootprint^[6].Y) THEN //Posizione Pinza - Metà ingombro - Offset sicurezza <= Ingombro colonna 
							Pinza_InIngombroColonne_Attuale := TRUE;
					ELSE
							Pinza_InIngombroColonne_Attuale := FALSE;
					END_IF
					(* Valuto la posizione futura - Missione di prelievo *)
					IF (Mission^.YPick - IngombroOttimizzatoX_InPuntoDiPrelievo/2 - OffsetSicurezza_Y <= WorkFootprint^[5].Y) OR //Posizione Pinza - Metà ingombro - Offset sicurezza <= Ingombro colonna 
						(Mission^.YPick + IngombroOttimizzatoX_InPuntoDiPrelievo/2 + OffsetSicurezza_Y >= WorkFootprint^[6].Y) THEN //Posizione Pinza - Metà ingombro - Offset sicurezza <= Ingombro colonna 
							Pinza_InIngombroColonne_Destinazione := TRUE;
					ELSE
							Pinza_InIngombroColonne_Destinazione := FALSE;
					END_IF
					
					(* Valuto la posizione futura - Missione di Deposito *)
					IF (Mission^.YPick - IngombroOttimizzatoX_InPuntoDiDeposito/2 - OffsetSicurezza_Y <= WorkFootprint^[5].Y) OR //Posizione Pinza - Metà ingombro - Offset sicurezza <= Ingombro colonna 
						(Mission^.YPick + IngombroOttimizzatoX_InPuntoDiDeposito/2 + OffsetSicurezza_Y >= WorkFootprint^[6].Y) THEN //Posizione Pinza - Metà ingombro - Offset sicurezza <= Ingombro colonna 
							Pinza_InIngombroColonne_Destinazione := TRUE;
					ELSE
							Pinza_InIngombroColonne_Destinazione := FALSE;
					END_IF
					
					(* Valuto la posizione attuale Y e la posizione di destinazione Y e l'ingombro massimo che posso avere durante il transito *)
					IF (Mission^.YPick - IngombroOttimizzatoY_InTransito/2 - OffsetSicurezza_Y <= WorkFootprint^[5].Y) OR //Posizione Pinza - Metà ingombro - Offset sicurezza <= Ingombro colonna 
						(Mission^.YPick + IngombroOttimizzatoY_InTransito/2 + OffsetSicurezza_Y >= WorkFootprint^[6].Y) THEN //Posizione Pinza - Metà ingombro - Offset sicurezza <= Ingombro colonna 
							Pinza_InIngombroColonne_Transito := TRUE;
					ELSE
							Pinza_InIngombroColonne_Transito := FALSE;
					END_IF
			END_CASE		
			(* Se sono in ingombro nella posizione attuale o nella posizione di destinazione, devo andare fuori-ingombro con la Y *)
			IF (Pinza_InIngombroColonne_Attuale OR Pinza_InIngombroColonne_Destinazione OR Pinza_InIngombroColonne_Transito) THEN 
				IF (AsseXInFinestraDiRiposo AND AsseYInFinestraDiRiposo AND AsseJInFinestraDiRiposo) THEN //Se sono in finestra di riposo con tutti gli assi non devo andare fuori-ingombro con la Y
					FuoriIngombroYNecessarioTMP := FALSE;
				ELSE
					FuoriIngombroYNecessarioTMP := TRUE;
				END_IF
			ELSE
				FuoriIngombroYNecessarioTMP := FALSE;
			END_IF
		END_IF
			
	WAMANAGER_CICLO_DEPOSITO_FALDA_END:
		CalcolaIngombro := TRUE;	

	WAMANAGER_CICLO_PACCO_INIT:
		CalcolaIngombro := TRUE;	
	
	WAMANAGER_CICLO_PRELIEVO_PACCO_RUN:
		
		IF CalcolaIngombro THEN
			CalcolaIngombro := FALSE;
			(* Definisco il tipo di area in cui si trova a lavorare il pallettizzatore *)
			AreaInLavoroPositiva := FALSE;
			AreaInLavoroNegativa := FALSE;
			AreaInLavoroPositivaNegativa := TRUE; 
			CASE Mission^.JPickVO OF
				(* Verticale *)
				0:	
					IF ModuleAx_X^.Ax^.AxRef^.NcToPlc.ActPos <= WorkFootprint^[5].X AND 
						WorkPickPoint^[Mission^.PPick].Xv <= WorkFootprint^[5].X THEN
							AreaInLavoroNegativa := TRUE;
					ELSIF ModuleAx_X^.Ax^.AxRef^.NcToPlc.ActPos >= WorkFootprint^[5].X AND 
						WorkPickPoint^[Mission^.PPick].Xv >= WorkFootprint^[5].X THEN
							AreaInLavoroPositiva := TRUE;
					ELSE
						AreaInLavoroPositiva := FALSE;
						AreaInLavoroNegativa := FALSE;
						AreaInLavoroPositivaNegativa := TRUE;
					END_IF
					
				(* Orrizontale *)
				1: 
					IF ModuleAx_X^.Ax^.AxRef^.NcToPlc.ActPos <= WorkFootprint^[5].X AND 
						WorkPickPoint^[Mission^.PPick].Xh <= WorkFootprint^[5].X THEN
							AreaInLavoroNegativa := TRUE;
					ELSIF ModuleAx_X^.Ax^.AxRef^.NcToPlc.ActPos >= (WorkFootprint^[5].X + WorkFootprint^[5].XDim) AND 
						WorkPickPoint^[Mission^.PPick].Xh >= (WorkFootprint^[5].X + WorkFootprint^[5].XDim) THEN
							AreaInLavoroPositiva := TRUE;
					ELSE
						AreaInLavoroPositiva := FALSE;
						AreaInLavoroNegativa := FALSE;
						AreaInLavoroPositivaNegativa := TRUE;
					END_IF
			END_CASE
			
			(**************************************************************************************************************************************************)
			(* Ingombro ottimizzato della pinza sul punto di prelievo *)
			(**************************************************************************************************************************************************)
			IngombroOttimizzatoX_InPuntoDiPrelievo := ABS(IngombroSuperficialePinzaMAX * SIN(deg_to_rad((ATAN(Larghezza/Lunghezza)*1/0.017+ Mission^.JPick))));
			IngombroOttimizzatoY_InPuntoDiPrelievo := ABS(IngombroSuperficialePinzaMAX * COS(deg_to_rad((ATAN(Larghezza/Lunghezza)*1/0.017+ Mission^.JPick))));
			(**************************************************************************************************************************************************)
			(* Ingombro ottimizzato della pinza sul punto di deposito *)
			(**************************************************************************************************************************************************)
			IngombroOttimizzatoX_InPuntoDiDeposito := ABS(IngombroSuperficialePinzaMAX * SIN(deg_to_rad((ATAN(Larghezza/Lunghezza)*1/0.017+ Mission^.JPlace))));
			IngombroOttimizzatoY_InPuntoDiDeposito := ABS(IngombroSuperficialePinzaMAX * COS(deg_to_rad((ATAN(Larghezza/Lunghezza)*1/0.017+ Mission^.JPlace))));
						
			(**************************************************************************************************************************************************)
			(**************************************************************************************************************************************************)
						
			(* Valuto la direzione della X *)
			DirezioneXPositiva := TFDirezioneAssePositiva(Posizione_Attuale:=ModuleAX_X^.Ax^.Status.ActPosition,Posizione_Finale:=Mission^.XPick);
			DirezioneXNegativa := NOT DirezioneXPositiva;
				
			(* Valuto se gli assi sono in finestra di prelievo *)
			AsseXInFinestraDiRiposo := TFAsseInFinestra(Posizione_Attuale:=ModuleAx_X^.Ax^.AxRef^.NcToPlc.ActPos,Posizione_Finale:=Mission^.XPick,FinestraDiControllo:=10);
			AsseYInFinestraDiRiposo := TFAsseInFinestra(Posizione_Attuale:=ModuleAx_Y^.Ax^.AxRef^.NcToPlc.ActPos,Posizione_Finale:=Mission^.YPick,FinestraDiControllo:=10);
			AsseJInFinestraDiRiposo := TFAsseInFinestra(Posizione_Attuale:=ModuleAx_J^.Ax^.AxRef^.NcToPlc.ActPos,Posizione_Finale:=Mission^.JPick,FinestraDiControllo:=5);
			(* Valuto se gli assi sono in finestra di destinazione *)
			AsseXInFinestraDiDestinazione := TFAsseInFinestra(Posizione_Attuale:=ModuleAx_X^.Ax^.AxRef^.NcToPlc.ActPos,Posizione_Finale:=Mission^.XPick,FinestraDiControllo:=10);
			AsseYInFinestraDiDestinazione := TFAsseInFinestra(Posizione_Attuale:=ModuleAx_Y^.Ax^.AxRef^.NcToPlc.ActPos,Posizione_Finale:=Mission^.YPick,FinestraDiControllo:=10);
			AsseJInFinestraDiDestinazione := TFAsseInFinestra(Posizione_Attuale:=ModuleAx_J^.Ax^.AxRef^.NcToPlc.ActPos,Posizione_Finale:=Mission^.JPick,FinestraDiControllo:=5);
			
			(**************************************************************************************************************************************************)
			(* Ingombro MASSIMO della pinza durante il transito *)
			(**************************************************************************************************************************************************)
			//Calcolo ingombro attuale
			IngombroOttimizzatoX_InTransito := ABS(IngombroSuperficialePinzaMAX * SIN(deg_to_rad((ATAN(Larghezza/Lunghezza)*1/0.017+ ModuleAx_J^.Ax^.AxRef^.NcToPlc.ActPos)))); //Ingombro Attuale direzione X
			IngombroOttimizzatoY_InTransito := ABS(IngombroSuperficialePinzaMAX * COS(deg_to_rad((ATAN(Larghezza/Lunghezza)*1/0.017+ ModuleAx_J^.Ax^.AxRef^.NcToPlc.ActPos)))); //Ingombro Attuale direzione Y		
			IF NOT AsseJInFinestraDiDestinazione THEN
				IF REAL_TO_INT(ModuleAx_J^.Ax^.AxRef^.NcToPlc.ActPos) <= REAL_TO_INT(Mission^.JPick) THEN
					FOR Angolo := REAL_TO_INT(ModuleAx_J^.Ax^.AxRef^.NcToPlc.ActPos) TO REAL_TO_INT(Mission^.JPick)  DO
						IF IngombroOttimizzatoX_InTransito < ABS(IngombroSuperficialePinzaMAX * SIN(deg_to_rad((ATAN(Larghezza/Lunghezza)*1/0.017+ Angolo)))) THEN
							IngombroOttimizzatoX_InTransito := ABS(IngombroSuperficialePinzaMAX * SIN(deg_to_rad((ATAN(Larghezza/Lunghezza)*1/0.017+ Angolo)))) ;
						END_IF
						IF IngombroOttimizzatoY_InTransito < ABS(IngombroSuperficialePinzaMAX * COS(deg_to_rad((ATAN(Larghezza/Lunghezza)*1/0.017+ Angolo)))) THEN
							IngombroOttimizzatoY_InTransito := ABS(IngombroSuperficialePinzaMAX * COS(deg_to_rad((ATAN(Larghezza/Lunghezza)*1/0.017+ Angolo))));
						END_IF
					END_FOR
				END_IF
			END_IF
		
			(* Valutazione colonne in base al verso del pallettizzatore *)
			CASE VERSO_PALLETTIZZATORE OF
				PALLETTIZZATORE_DX:	// Colonna 6:DX, 5:SX
					(* Valuto la posizione attuale *)
					IF (ModuleAX_Y^.Ax^.Status.ActPosition - IngombroY/2 - OffsetSicurezza_Y <= WorkFootprint^[6].Y) OR //Posizione Pinza - Metà ingombro - Offset sicurezza <= Ingombro colonna 
						(ModuleAX_Y^.Ax^.Status.ActPosition + IngombroY/2 + OffsetSicurezza_Y >= WorkFootprint^[5].Y) THEN //Posizione Pinza - Metà ingombro - Offset sicurezza <= Ingombro colonna 
							Pinza_InIngombroColonne_Attuale := TRUE;
					ELSE
							Pinza_InIngombroColonne_Attuale := FALSE;
					END_IF
					(* Valuto la posizione futura - Missione di prelievo *)
					IF (Mission^.YPick - IngombroOttimizzatoX_InPuntoDiPrelievo/2 - OffsetSicurezza_Y <= WorkFootprint^[6].Y) OR //Posizione Pinza - Metà ingombro - Offset sicurezza <= Ingombro colonna 
						(Mission^.YPick + IngombroOttimizzatoX_InPuntoDiPrelievo/2 + OffsetSicurezza_Y >= WorkFootprint^[5].Y) THEN //Posizione Pinza - Metà ingombro - Offset sicurezza <= Ingombro colonna 
							Pinza_InIngombroColonne_Destinazione := TRUE;
					ELSE
							Pinza_InIngombroColonne_Destinazione := FALSE;
					END_IF
					
					(* Valuto la posizione futura - Missione di Deposito *)
					IF (Mission^.YPick - IngombroOttimizzatoX_InPuntoDiDeposito/2 - OffsetSicurezza_Y <= WorkFootprint^[6].Y) OR //Posizione Pinza - Metà ingombro - Offset sicurezza <= Ingombro colonna 
						(Mission^.YPick + IngombroOttimizzatoX_InPuntoDiDeposito/2 + OffsetSicurezza_Y >= WorkFootprint^[5].Y) THEN //Posizione Pinza - Metà ingombro - Offset sicurezza <= Ingombro colonna 
							Pinza_InIngombroColonne_Destinazione := TRUE;
					ELSE
							Pinza_InIngombroColonne_Destinazione := FALSE;
					END_IF
					
					(* Valuto la posizione attuale Y e la posizione di destinazione Y e l'ingombro massimo che posso avere durante il transito *)
					IF (Mission^.YPick - IngombroOttimizzatoY_InTransito/2 - OffsetSicurezza_Y <= WorkFootprint^[6].Y) OR //Posizione Pinza - Metà ingombro - Offset sicurezza <= Ingombro colonna 
						(Mission^.YPick + IngombroOttimizzatoY_InTransito/2 + OffsetSicurezza_Y >= WorkFootprint^[5].Y) THEN //Posizione Pinza - Metà ingombro - Offset sicurezza <= Ingombro colonna 
							Pinza_InIngombroColonne_Transito := TRUE;
					ELSE
							Pinza_InIngombroColonne_Transito := FALSE;
					END_IF
						
				PALLETTIZZATORE_SX: // Colonna 6:SX, 5:DX
					(* Valuto la posizione attuale *)
					IF (ModuleAX_Y^.Ax^.Status.ActPosition - IngombroY/2 - OffsetSicurezza_Y <= WorkFootprint^[5].Y) OR //Posizione Pinza - Metà ingombro - Offset sicurezza <= Ingombro colonna 
						(ModuleAX_Y^.Ax^.Status.ActPosition + IngombroY/2 + OffsetSicurezza_Y >= WorkFootprint^[6].Y) THEN //Posizione Pinza - Metà ingombro - Offset sicurezza <= Ingombro colonna 
							Pinza_InIngombroColonne_Attuale := TRUE;
					ELSE
							Pinza_InIngombroColonne_Attuale := FALSE;
					END_IF
					(* Valuto la posizione futura - Missione di prelievo *)
					IF (Mission^.YPick - IngombroOttimizzatoX_InPuntoDiPrelievo/2 - OffsetSicurezza_Y <= WorkFootprint^[5].Y) OR //Posizione Pinza - Metà ingombro - Offset sicurezza <= Ingombro colonna 
						(Mission^.YPick + IngombroOttimizzatoX_InPuntoDiPrelievo/2 + OffsetSicurezza_Y >= WorkFootprint^[6].Y) THEN //Posizione Pinza - Metà ingombro - Offset sicurezza <= Ingombro colonna 
							Pinza_InIngombroColonne_Destinazione := TRUE;
					ELSE
							Pinza_InIngombroColonne_Destinazione := FALSE;
					END_IF
					
					(* Valuto la posizione futura - Missione di Deposito *)
					IF (Mission^.YPick - IngombroOttimizzatoX_InPuntoDiDeposito/2 - OffsetSicurezza_Y <= WorkFootprint^[5].Y) OR //Posizione Pinza - Metà ingombro - Offset sicurezza <= Ingombro colonna 
						(Mission^.YPick + IngombroOttimizzatoX_InPuntoDiDeposito/2 + OffsetSicurezza_Y >= WorkFootprint^[6].Y) THEN //Posizione Pinza - Metà ingombro - Offset sicurezza <= Ingombro colonna 
							Pinza_InIngombroColonne_Destinazione := TRUE;
					ELSE
							Pinza_InIngombroColonne_Destinazione := FALSE;
					END_IF
					
					(* Valuto la posizione attuale Y e la posizione di destinazione Y e l'ingombro massimo che posso avere durante il transito *)
					IF (Mission^.YPick - IngombroOttimizzatoY_InTransito/2 - OffsetSicurezza_Y <= WorkFootprint^[5].Y) OR //Posizione Pinza - Metà ingombro - Offset sicurezza <= Ingombro colonna 
						(Mission^.YPick + IngombroOttimizzatoY_InTransito/2 + OffsetSicurezza_Y >= WorkFootprint^[6].Y) THEN //Posizione Pinza - Metà ingombro - Offset sicurezza <= Ingombro colonna 
							Pinza_InIngombroColonne_Transito := TRUE;
					ELSE
							Pinza_InIngombroColonne_Transito := FALSE;
					END_IF
			END_CASE		
			(* Se sono in ingombro nella posizione attuale o nella posizione di destinazione, devo andare fuori-ingombro con la Y *)
			IF (Pinza_InIngombroColonne_Attuale OR Pinza_InIngombroColonne_Destinazione OR Pinza_InIngombroColonne_Transito) THEN 
				IF (AsseXInFinestraDiRiposo AND AsseYInFinestraDiRiposo AND AsseJInFinestraDiRiposo) THEN //Se sono in finestra di riposo con tutti gli assi non devo andare fuori-ingombro con la Y
					FuoriIngombroYNecessarioTMP := FALSE;
				ELSE
					FuoriIngombroYNecessarioTMP := TRUE;
				END_IF
			ELSE
				FuoriIngombroYNecessarioTMP := FALSE;
			END_IF
		END_IF
	WAMANAGER_CICLO_PRELIEVO_PACCO_END:
		CalcolaIngombro := TRUE;	
		
	WAMANAGER_CICLO_DEPOSITO_PACCO_RUN:
	
		IF CalcolaIngombro THEN
			CalcolaIngombro := FALSE;
			(* Definisco il tipo di area in cui si trova a lavorare il pallettizzatore *)
			AreaInLavoroPositiva := FALSE;
			AreaInLavoroNegativa := FALSE;
			AreaInLavoroPositivaNegativa := FALSE; 
			
			IF ModuleAx_X^.Ax^.AxRef^.NcToPlc.ActPos >= (WorkFootprint^[5].X + WorkFootprint^[5].XDim) AND 	//se la piazzola di prelievo ha quota maggiore rispetto le colonne centrali
				WorkArea^[Mission^.PPlace].X >= (WorkFootprint^[5].X + WorkFootprint^[5].XDim)  THEN //la piazzola di deposito è nella campata positiva
					AreaInLavoroPositiva := TRUE;
			ELSIF ModuleAx_X^.Ax^.AxRef^.NcToPlc.ActPos <= WorkFootprint^[5].X AND 	//se la piazzola di prelievo ha quota maggiore della piazzola di deposito e
				WorkArea^[Mission^.PPlace].X <= WorkFootprint^[5].X  THEN //la piazzola di deposito è nella campata negativa
					AreaInLavoroNegativa := TRUE;
			ELSE
				AreaInLavoroPositiva := FALSE;
				AreaInLavoroNegativa := FALSE;
				AreaInLavoroPositivaNegativa := TRUE;
			END_IF
			
			(**************************************************************************************************************************************************)
			(* Ingombro ottimizzato della pinza sul punto di prelievo *)
			(**************************************************************************************************************************************************)
			IngombroOttimizzatoX_InPuntoDiPrelievo := ABS(IngombroSuperficialePinzaMAX * SIN(deg_to_rad((ATAN(Larghezza/Lunghezza)*1/0.017+ Mission^.JPick))));
			IngombroOttimizzatoY_InPuntoDiPrelievo := ABS(IngombroSuperficialePinzaMAX * COS(deg_to_rad((ATAN(Larghezza/Lunghezza)*1/0.017+ Mission^.JPick))));
			(**************************************************************************************************************************************************)
			(* Ingombro ottimizzato della pinza sul punto di deposito *)
			(**************************************************************************************************************************************************)
			IngombroOttimizzatoX_InPuntoDiDeposito := ABS(IngombroSuperficialePinzaMAX * SIN(deg_to_rad((ATAN(Larghezza/Lunghezza)*1/0.017+ Mission^.JPlace))));
			IngombroOttimizzatoY_InPuntoDiDeposito := ABS(IngombroSuperficialePinzaMAX * COS(deg_to_rad((ATAN(Larghezza/Lunghezza)*1/0.017+ Mission^.JPlace))));
						
			(**************************************************************************************************************************************************)
			(**************************************************************************************************************************************************)
						
			(* Valuto la direzione della X *)
			DirezioneXPositiva := TFDirezioneAssePositiva(Posizione_Attuale:=ModuleAX_X^.Ax^.Status.ActPosition,Posizione_Finale:=Mission^.XPick);
			DirezioneXNegativa := NOT DirezioneXPositiva;
				
			(* Valuto se gli assi sono in finestra di prelievo *)
			AsseXInFinestraDiRiposo := TFAsseInFinestra(Posizione_Attuale:=ModuleAx_X^.Ax^.AxRef^.NcToPlc.ActPos,Posizione_Finale:=Mission^.XPick,FinestraDiControllo:=10);
			AsseYInFinestraDiRiposo := TFAsseInFinestra(Posizione_Attuale:=ModuleAx_Y^.Ax^.AxRef^.NcToPlc.ActPos,Posizione_Finale:=Mission^.YPick,FinestraDiControllo:=10);
			AsseJInFinestraDiRiposo := TFAsseInFinestra(Posizione_Attuale:=ModuleAx_J^.Ax^.AxRef^.NcToPlc.ActPos,Posizione_Finale:=Mission^.JPick,FinestraDiControllo:=5);
			(* Valuto se gli assi sono in finestra di destinazione *)
			AsseXInFinestraDiDestinazione := TFAsseInFinestra(Posizione_Attuale:=ModuleAx_X^.Ax^.AxRef^.NcToPlc.ActPos,Posizione_Finale:=Mission^.XPick,FinestraDiControllo:=10);
			AsseYInFinestraDiDestinazione := TFAsseInFinestra(Posizione_Attuale:=ModuleAx_Y^.Ax^.AxRef^.NcToPlc.ActPos,Posizione_Finale:=Mission^.YPick,FinestraDiControllo:=10);
			AsseJInFinestraDiDestinazione := TFAsseInFinestra(Posizione_Attuale:=ModuleAx_J^.Ax^.AxRef^.NcToPlc.ActPos,Posizione_Finale:=Mission^.JPick,FinestraDiControllo:=5);
			
			(**************************************************************************************************************************************************)
			(* Ingombro MASSIMO della pinza durante il transito *)
			(**************************************************************************************************************************************************)
			//Calcolo ingombro attuale
			IngombroOttimizzatoX_InTransito := ABS(IngombroSuperficialePinzaMAX * SIN(deg_to_rad((ATAN(Larghezza/Lunghezza)*1/0.017+ ModuleAx_J^.Ax^.AxRef^.NcToPlc.ActPos)))); //Ingombro Attuale direzione X
			IngombroOttimizzatoY_InTransito := ABS(IngombroSuperficialePinzaMAX * COS(deg_to_rad((ATAN(Larghezza/Lunghezza)*1/0.017+ ModuleAx_J^.Ax^.AxRef^.NcToPlc.ActPos)))); //Ingombro Attuale direzione Y		
			IF NOT AsseJInFinestraDiDestinazione THEN
				IF REAL_TO_INT(ModuleAx_J^.Ax^.AxRef^.NcToPlc.ActPos) <= REAL_TO_INT(Mission^.JPick) THEN
					FOR Angolo := REAL_TO_INT(ModuleAx_J^.Ax^.AxRef^.NcToPlc.ActPos) TO REAL_TO_INT(Mission^.JPick)  DO
						IF IngombroOttimizzatoX_InTransito < ABS(IngombroSuperficialePinzaMAX * SIN(deg_to_rad((ATAN(Larghezza/Lunghezza)*1/0.017+ Angolo)))) THEN
							IngombroOttimizzatoX_InTransito := ABS(IngombroSuperficialePinzaMAX * SIN(deg_to_rad((ATAN(Larghezza/Lunghezza)*1/0.017+ Angolo)))) ;
						END_IF
						IF IngombroOttimizzatoY_InTransito < ABS(IngombroSuperficialePinzaMAX * COS(deg_to_rad((ATAN(Larghezza/Lunghezza)*1/0.017+ Angolo)))) THEN
							IngombroOttimizzatoY_InTransito := ABS(IngombroSuperficialePinzaMAX * COS(deg_to_rad((ATAN(Larghezza/Lunghezza)*1/0.017+ Angolo))));
						END_IF
					END_FOR
				END_IF
			END_IF
		
			(* Valutazione colonne in base al verso del pallettizzatore *)
			CASE VERSO_PALLETTIZZATORE OF
				PALLETTIZZATORE_DX:	// Colonna 6:DX, 5:SX
					(* Valuto la posizione attuale *)
					IF (ModuleAX_Y^.Ax^.Status.ActPosition - IngombroY/2 - OffsetSicurezza_Y <= WorkFootprint^[6].Y) OR //Posizione Pinza - Metà ingombro - Offset sicurezza <= Ingombro colonna 
						(ModuleAX_Y^.Ax^.Status.ActPosition + IngombroY/2 + OffsetSicurezza_Y >= WorkFootprint^[5].Y) THEN //Posizione Pinza - Metà ingombro - Offset sicurezza <= Ingombro colonna 
							Pinza_InIngombroColonne_Attuale := TRUE;
					ELSE
							Pinza_InIngombroColonne_Attuale := FALSE;
					END_IF
					(* Valuto la posizione futura - Missione di prelievo *)
					IF (Mission^.YPick - IngombroOttimizzatoX_InPuntoDiPrelievo/2 - OffsetSicurezza_Y <= WorkFootprint^[6].Y) OR //Posizione Pinza - Metà ingombro - Offset sicurezza <= Ingombro colonna 
						(Mission^.YPick + IngombroOttimizzatoX_InPuntoDiPrelievo/2 + OffsetSicurezza_Y >= WorkFootprint^[5].Y) THEN //Posizione Pinza - Metà ingombro - Offset sicurezza <= Ingombro colonna 
							Pinza_InIngombroColonne_Destinazione := TRUE;
					ELSE
							Pinza_InIngombroColonne_Destinazione := FALSE;
					END_IF
					
					(* Valuto la posizione futura - Missione di Deposito *)
					IF (Mission^.YPick - IngombroOttimizzatoX_InPuntoDiDeposito/2 - OffsetSicurezza_Y <= WorkFootprint^[6].Y) OR //Posizione Pinza - Metà ingombro - Offset sicurezza <= Ingombro colonna 
						(Mission^.YPick + IngombroOttimizzatoX_InPuntoDiDeposito/2 + OffsetSicurezza_Y >= WorkFootprint^[5].Y) THEN //Posizione Pinza - Metà ingombro - Offset sicurezza <= Ingombro colonna 
							Pinza_InIngombroColonne_Destinazione := TRUE;
					ELSE
							Pinza_InIngombroColonne_Destinazione := FALSE;
					END_IF
					
					(* Valuto la posizione attuale Y e la posizione di destinazione Y e l'ingombro massimo che posso avere durante il transito *)
					IF (Mission^.YPick - IngombroOttimizzatoY_InTransito/2 - OffsetSicurezza_Y <= WorkFootprint^[6].Y) OR //Posizione Pinza - Metà ingombro - Offset sicurezza <= Ingombro colonna 
						(Mission^.YPick + IngombroOttimizzatoY_InTransito/2 + OffsetSicurezza_Y >= WorkFootprint^[5].Y) THEN //Posizione Pinza - Metà ingombro - Offset sicurezza <= Ingombro colonna 
							Pinza_InIngombroColonne_Transito := TRUE;
					ELSE
							Pinza_InIngombroColonne_Transito := FALSE;
					END_IF
						
				PALLETTIZZATORE_SX: // Colonna 6:SX, 5:DX
					(* Valuto la posizione attuale *)
					IF (ModuleAX_Y^.Ax^.Status.ActPosition - IngombroY/2 - OffsetSicurezza_Y <= WorkFootprint^[5].Y) OR //Posizione Pinza - Metà ingombro - Offset sicurezza <= Ingombro colonna 
						(ModuleAX_Y^.Ax^.Status.ActPosition + IngombroY/2 + OffsetSicurezza_Y >= WorkFootprint^[6].Y) THEN //Posizione Pinza - Metà ingombro - Offset sicurezza <= Ingombro colonna 
							Pinza_InIngombroColonne_Attuale := TRUE;
					ELSE
							Pinza_InIngombroColonne_Attuale := FALSE;
					END_IF
					(* Valuto la posizione futura - Missione di prelievo *)
					IF (Mission^.YPick - IngombroOttimizzatoX_InPuntoDiPrelievo/2 - OffsetSicurezza_Y <= WorkFootprint^[5].Y) OR //Posizione Pinza - Metà ingombro - Offset sicurezza <= Ingombro colonna 
						(Mission^.YPick + IngombroOttimizzatoX_InPuntoDiPrelievo/2 + OffsetSicurezza_Y >= WorkFootprint^[6].Y) THEN //Posizione Pinza - Metà ingombro - Offset sicurezza <= Ingombro colonna 
							Pinza_InIngombroColonne_Destinazione := TRUE;
					ELSE
							Pinza_InIngombroColonne_Destinazione := FALSE;
					END_IF
					
					(* Valuto la posizione futura - Missione di Deposito *)
					IF (Mission^.YPick - IngombroOttimizzatoX_InPuntoDiDeposito/2 - OffsetSicurezza_Y <= WorkFootprint^[5].Y) OR //Posizione Pinza - Metà ingombro - Offset sicurezza <= Ingombro colonna 
						(Mission^.YPick + IngombroOttimizzatoX_InPuntoDiDeposito/2 + OffsetSicurezza_Y >= WorkFootprint^[6].Y) THEN //Posizione Pinza - Metà ingombro - Offset sicurezza <= Ingombro colonna 
							Pinza_InIngombroColonne_Destinazione := TRUE;
					ELSE
							Pinza_InIngombroColonne_Destinazione := FALSE;
					END_IF
					
					(* Valuto la posizione attuale Y e la posizione di destinazione Y e l'ingombro massimo che posso avere durante il transito *)
					IF (Mission^.YPick - IngombroOttimizzatoY_InTransito/2 - OffsetSicurezza_Y <= WorkFootprint^[5].Y) OR //Posizione Pinza - Metà ingombro - Offset sicurezza <= Ingombro colonna 
						(Mission^.YPick + IngombroOttimizzatoY_InTransito/2 + OffsetSicurezza_Y >= WorkFootprint^[6].Y) THEN //Posizione Pinza - Metà ingombro - Offset sicurezza <= Ingombro colonna 
							Pinza_InIngombroColonne_Transito := TRUE;
					ELSE
							Pinza_InIngombroColonne_Transito := FALSE;
					END_IF
			END_CASE		
			(* Se sono in ingombro nella posizione attuale o nella posizione di destinazione, devo andare fuori-ingombro con la Y *)
			IF (Pinza_InIngombroColonne_Attuale OR Pinza_InIngombroColonne_Destinazione OR Pinza_InIngombroColonne_Transito) THEN 
				IF (AsseXInFinestraDiRiposo AND AsseYInFinestraDiRiposo AND AsseJInFinestraDiRiposo) THEN //Se sono in finestra di riposo con tutti gli assi non devo andare fuori-ingombro con la Y
					FuoriIngombroYNecessarioTMP := FALSE;
				ELSE
					FuoriIngombroYNecessarioTMP := TRUE;
				END_IF
			ELSE
				FuoriIngombroYNecessarioTMP := FALSE;
			END_IF
		END_IF
		
	WAMANAGER_CICLO_DEPOSITO_PACCO_END:
		CalcolaIngombro := TRUE;	
	
END_CASE

TFCalcoliFuoriIngombriColonne := TRUE;

END_FUNCTION

// ---- POUs/TFPalletizerDataTF/NON_USATE/TFNumeroPacchiSuLinea_OLD.TcPOU
FUNCTION TFNumeroPacchiSuLinea_OLD : UINT
VAR_INPUT
	HandlingPackTable : POINTER TO TFHandlingPackTable;
END_VAR
VAR
	i : UINT;
END_VAR

TFNumeroPacchiSuLinea := 0; 

FOR i:= 1 TO MAXHANDLINGPACK DO
	IF HandlingPackTable^.Table[i,1].PP THEN
		TFNumeroPacchiSuLinea := TFNumeroPacchiSuLinea +1;
	END_IF
END_FOR

END_FUNCTION

// ---- POUs/TFPalletizerDataTF/NON_USATE/TFNumeroUltimi_N_TrasportiOccupati_OLD.TcPOU
FUNCTION TFNumeroUltimi_N_TrasportiOccupati_OLD : UINT // Restituisce il numero di trasporti occupati, dall'ultimo all' n-esimo
VAR_INPUT
	HandlingPackTable : POINTER TO TFHandlingPackTable;
	NTrasportiDaControllare : UINT;
END_VAR
VAR
	i : UINT;
END_VAR

TFNumeroUltimi_N_TrasportiOccupati := 0; 

FOR i:= MAXHANDLINGPACK TO (MAXHANDLINGPACK - NTrasportiDaControllare - 1) BY -1 DO
	IF i >= NTrasportiDaControllare THEN
		IF HandlingPackTable^.Table[i,1].PP THEN
			TFNumeroUltimi_N_TrasportiOccupati := TFNumeroUltimi_N_TrasportiOccupati +1;
		END_IF
	ELSE
		RETURN;
	END_IF
END_FOR

END_FUNCTION

// ---- POUs/TFPalletizerDataTF/NON_USATE/TFPalletizer_CalcolaCoordinataPrelievo_WorkArea.TcPOU
FUNCTION_BLOCK TFPalletizer_CalcolaCoordinataPrelievo_WorkArea
VAR_INPUT
	WorkArea 		: POINTER TO ARRAY [1..MAXAREA] OF TFMachinePalletizer_WorkArea;
	WorkAreaState 	: POINTER TO ARRAY [1..MAXAREA] OF TFMachinePalletizer_WorkAreaState;
	WorkAreaOffset	: POINTER TO ARRAY [1..MAXAREA] OF TFMachinePalletizer_WorkAreaOffset;
	
	Forming 		: POINTER TO ARRAY [1..MAXFORMING] OF TFMachinePalletizer_Forming;
	Pallet 			: POINTER TO ARRAY [1..MAXPALLET] OF TFMachinePalletizer_Pallet;
	Layer 			: POINTER TO ARRAY [1..MAXLAYER] OF TFMachinePalletizer_Layer;
	Mission 		: POINTER TO TFMachinePalletizer_Mission;
	
	WADiPrelievo				: UINT;
	NLastraDaPrelevare			: UINT;
END_VAR
VAR_OUTPUT
	Errore : TFError_WAM;
END_VAR
VAR
END_VAR

Errore.Code := 0;

CASE DISPOSIZIONE_FTC_WA OF
	FTC_PRESENZA_ANGOLO_DX :
		(*******************************************************************************************************************)
									(* Deposito LASTRA con rotazione piano >90° e < 180°*)
		(*******************************************************************************************************************)																		
		IF Forming^[WorkAreaState^[WADiPrelievo].F].PackXP[NLastraDaPrelevare].J > 90 THEN
			
			Mission^.XPick	:= WorkArea^[WADiPrelievo].X + WorkAreaOffset^[WADiPrelievo].X -  																																					(* Quota X del Cavaletto *)	
								Forming^[WorkAreaState^[WADiPrelievo].F].PackXP[NLastraDaPrelevare].X+	
								Pallet^[Forming^[WorkAreaState^[WADiPrelievo].F].Pallet].OFSDE_X180;	
		
			Mission^.YPick := WorkArea^[WADiPrelievo].Y + WorkAreaOffset^[WADiPrelievo].Y - 																																				(* Quota Y del Cavaletto *)		
								Forming^[WorkAreaState^[WADiPrelievo].F].PackXP[NLastraDaPrelevare].Y + 
								Pallet^[Forming^[WorkAreaState^[WADiPrelievo].F].Pallet].OFSDE_Y180;
								
			Mission^.ZPick	:= WorkArea^[WADiPrelievo].Z + WorkAreaOffset^[WADiPrelievo].Z +
								Forming^[WorkAreaState^[WADiPrelievo].F].PackXP[NLastraDaPrelevare].Z +	
								Pallet^[Forming^[WorkAreaState^[WADiPrelievo].F].Pallet].OFSDE_Z180;
					
			Mission^.JPick	:= Forming^[WorkAreaState^[WADiPrelievo].F].PackXP[WorkAreaState^[WADiPrelievo].PackPointer].J +	
								Pallet^[Forming^[WorkAreaState^[WADiPrelievo].F].Pallet].OFSDE_J180;
								
		(*******************************************************************************************************************)						
									(* Deposito LASTRA con rotazione piano < 90° e >0°*)	
		(*******************************************************************************************************************)							
		ELSIF Forming^[WorkAreaState^[WADiPrelievo].F].PackXP[WorkAreaState^[WADiPrelievo].PackPointer].J < 90 THEN
			
			Mission^.XPick	:= WorkArea^[WADiPrelievo].X + WorkAreaOffset^[WADiPrelievo].X - 																																					(* Quota X del Cavaletto *)	
								Forming^[WorkAreaState^[WADiPrelievo].F].PackXP[NLastraDaPrelevare].X+	
								Pallet^[Forming^[WorkAreaState^[WADiPrelievo].F].Pallet].OFSDE_X0;
								
			Mission^.YPick := WorkArea^[WADiPrelievo].Y + WorkAreaOffset^[WADiPrelievo].Y + 																																				(* Quota Y del Cavaletto *)						
								Forming^[WorkAreaState^[WADiPrelievo].F].PackXP[NLastraDaPrelevare].Y +
								Pallet^[Forming^[WorkAreaState^[WADiPrelievo].F].Pallet].OFSDE_Y0;
								
			Mission^.ZPick	:= WorkArea^[WADiPrelievo].Z + WorkAreaOffset^[WADiPrelievo].Z +
								Forming^[WorkAreaState^[WADiPrelievo].F].PackXP[NLastraDaPrelevare].Z +	
								Pallet^[Forming^[WorkAreaState^[WADiPrelievo].F].Pallet].OFSDE_Z0;
					
			Mission^.JPick	:= Forming^[WorkAreaState^[WADiPrelievo].F].PackXP[1].J +	
								Pallet^[Forming^[WorkAreaState^[WADiPrelievo].F].Pallet].OFSDE_J0;
		(*******************************************************************************************************************)						
									(* Deposito LASTRA in cassa con rotazione piano = 90° *)
		(*******************************************************************************************************************)
		ELSE
			
			Mission^.XPick	:= WorkArea^[WADiPrelievo].X + WorkAreaOffset^[WADiPrelievo].X + 																																					(* Quota X del Cavaletto *)	
								Forming^[WorkAreaState^[WADiPrelievo].F].PackXP[NLastraDaPrelevare].X+	
								Pallet^[Forming^[WorkAreaState^[WADiPrelievo].F].Pallet].OFSDE_X90;
								
			Mission^.YPick := WorkArea^[WADiPrelievo].Y + WorkAreaOffset^[WADiPrelievo].Y + 																																				(* Quota Y del Cavaletto *)						
								Forming^[WorkAreaState^[WADiPrelievo].F].PackXP[NLastraDaPrelevare].Y + 
								Pallet^[Forming^[WorkAreaState^[WADiPrelievo].F].Pallet].OFSDE_Y90;
									
			Mission^.ZPick	:= WorkArea^[WADiPrelievo].Z + WorkAreaOffset^[WADiPrelievo].Z +
								Forming^[WorkAreaState^[WADiPrelievo].F].PackXP[NLastraDaPrelevare].Z +	
								Pallet^[Forming^[WorkAreaState^[WADiPrelievo].F].Pallet].OFSDE_Z90;
								
			Mission^.JPick	:= Forming^[WorkAreaState^[WADiPrelievo].F].PackXP[NLastraDaPrelevare].J +	
								Pallet^[Forming^[WorkAreaState^[WADiPrelievo].F].Pallet].OFSDE_J90;
		END_IF
		
	FTC_PRESENZA_CENTRALE :
		(*******************************************************************************************************************)
									(* Deposito LASTRA con rotazione piano >90° e < 180°*)
		(*******************************************************************************************************************)																		
		IF Forming^[WorkAreaState^[WADiPrelievo].F].PackXP[WorkAreaState^[WADiPrelievo].PackPointer].J > 90 THEN
			
			Mission^.XPick	:= WorkArea^[WADiPrelievo].X + WorkAreaOffset^[WADiPrelievo].X + 																																					(* Quota X del Cavaletto *)	
								Forming^[WorkAreaState^[WADiPrelievo].F].PackXP[NLastraDaPrelevare].X +
								Pallet^[Forming^[WorkAreaState^[WADiPrelievo].F].Pallet].OFSDE_X180;		
		
			Mission^.YPick := WorkArea^[WADiPrelievo].Y + WorkAreaOffset^[WADiPrelievo].Y - 																																				(* Quota Y del Cavaletto *)		
								Forming^[WorkAreaState^[WADiPrelievo].F].PackXP[NLastraDaPrelevare].Y +
								Pallet^[Forming^[WorkAreaState^[WADiPrelievo].F].Pallet].OFSDE_Y180;
									
			Mission^.ZPick	:= WorkArea^[WADiPrelievo].Z + WorkAreaOffset^[WADiPrelievo].Z +
								Forming^[WorkAreaState^[WADiPrelievo].F].PackXP[NLastraDaPrelevare].Z +	
								Pallet^[Forming^[WorkAreaState^[WADiPrelievo].F].Pallet].OFSDE_Z180;
					
			Mission^.JPick	:= Forming^[WorkAreaState^[WADiPrelievo].F].PackXP[WorkAreaState^[WADiPrelievo].PackPointer].J +	
								Pallet^[Forming^[WorkAreaState^[WADiPrelievo].F].Pallet].OFSDE_J180;
								
		(*******************************************************************************************************************)						
									(* Deposito LASTRA con rotazione piano < 90° e >0°*)	
		(*******************************************************************************************************************)							
		ELSIF Forming^[WorkAreaState^[WADiPrelievo].F].PackXP[NLastraDaPrelevare].J < 90 THEN
			
			Mission^.XPick	:= WorkArea^[WADiPrelievo].X + WorkAreaOffset^[WADiPrelievo].X + 																																					(* Quota X del Cavaletto *)	
								Forming^[WorkAreaState^[WADiPrelievo].F].PackXP[NLastraDaPrelevare].X +
								Pallet^[Forming^[WorkAreaState^[WADiPrelievo].F].Pallet].OFSDE_X0;
								
			Mission^.YPick := WorkArea^[WADiPrelievo].Y + WorkAreaOffset^[WADiPrelievo].X + 																	(* Quota di deposito Y Ultima Lastra Depositata *)
								Pallet^[Forming^[WorkAreaState^[WADiPrelievo].F].Pallet].OFSDE_Y0;
									
			Mission^.ZPick	:= WorkArea^[WADiPrelievo].Z + WorkAreaOffset^[WADiPrelievo].Z +
								Forming^[WorkAreaState^[WADiPrelievo].F].PackXP[NLastraDaPrelevare].Z +	
								Pallet^[Forming^[WorkAreaState^[WADiPrelievo].F].Pallet].OFSDE_Z0;
					
			Mission^.JPick	:= Forming^[WorkAreaState^[WADiPrelievo].F].PackXP[NLastraDaPrelevare].J +	
								Pallet^[Forming^[WorkAreaState^[WADiPrelievo].F].Pallet].OFSDE_J0;
		(*******************************************************************************************************************)						
									(* Deposito su LASTRA in cassa con rotazione piano = 90° *)
		(*******************************************************************************************************************)
		ELSE
			Mission^.XPick	:= WorkArea^[WADiPrelievo].X + WorkAreaOffset^[WADiPrelievo].X + 																																					(* Quota X del Cavaletto *)	
								Forming^[WorkAreaState^[WADiPrelievo].F].PackXP[NLastraDaPrelevare].X+	
								Pallet^[Forming^[WorkAreaState^[WADiPrelievo].F].Pallet].OFSDE_X90;
								
			Mission^.YPick := WorkArea^[WADiPrelievo].Y + WorkAreaOffset^[WADiPrelievo].Y + 																																				(* Quota Y del Cavaletto *)						
								Forming^[WorkAreaState^[WADiPrelievo].F].PackXP[NLastraDaPrelevare].Y + 																	(* Quota di deposito Y Ultima Lastra Depositata *)
								Pallet^[Forming^[WorkAreaState^[WADiPrelievo].F].Pallet].OFSDE_Y90;
									
			Mission^.ZPick	:= WorkArea^[WADiPrelievo].Z + WorkAreaOffset^[WADiPrelievo].Z +
								Forming^[WorkAreaState^[WADiPrelievo].F].PackXP[1].Z +	
								Pallet^[Forming^[WorkAreaState^[WADiPrelievo].F].Pallet].OFSDE_Z90;
			Mission^.JPick	:= Forming^[WorkAreaState^[WADiPrelievo].F].PackXP[NLastraDaPrelevare].J +	
								Pallet^[Forming^[WorkAreaState^[WADiPrelievo].F].Pallet].OFSDE_J90;
		END_IF
		
	FTC_PRESENZA_ANGOLO_SX :
		(*******************************************************************************************************************)
									(* Deposito su LASTRA con rotazione piano >90° e < 180°*)
		(*******************************************************************************************************************)
		IF Forming^[WorkAreaState^[WADiPrelievo].F].PackXP[NLastraDaPrelevare].J > 90 THEN
			
			Mission^.XPick	:= WorkArea^[WADiPrelievo].X + WorkAreaOffset^[WADiPrelievo].X + 																																					(* Quota X del Cavaletto *)	
								Forming^[WorkAreaState^[WADiPrelievo].F].PackXP[NLastraDaPrelevare].X +
								Pallet^[Forming^[WorkAreaState^[WADiPrelievo].F].Pallet].OFSDE_X180;	
		
			Mission^.YPick := WorkArea^[WADiPrelievo].Y + WorkAreaOffset^[WADiPrelievo].Y - 																																				(* Quota Y del Cavaletto *)		
								Forming^[WorkAreaState^[WADiPrelievo].F].PackXP[NLastraDaPrelevare].Y +
								Pallet^[Forming^[WorkAreaState^[WADiPrelievo].F].Pallet].OFSDE_Y180;
									
			Mission^.ZPick	:= WorkArea^[WADiPrelievo].Z + WorkAreaOffset^[WADiPrelievo].Z +
								Forming^[WorkAreaState^[WADiPrelievo].F].PackXP[NLastraDaPrelevare].Z +	
								Pallet^[Forming^[WorkAreaState^[WADiPrelievo].F].Pallet].OFSDE_Z180;
					
			Mission^.JPick	:= Forming^[WorkAreaState^[WADiPrelievo].F].PackXP[NLastraDaPrelevare].J +	
								Pallet^[Forming^[WorkAreaState^[WADiPrelievo].F].Pallet].OFSDE_J180;
		(*******************************************************************************************************************)						
									(* Deposito su LASTRA con rotazione piano < 90° e >0°*)	
		(*******************************************************************************************************************)
		ELSIF Forming^[WorkAreaState^[WADiPrelievo].F].PackXP[WorkAreaState^[WADiPrelievo].PackPointer].J < 90 THEN
			
			Mission^.XPick	:= WorkArea^[WADiPrelievo].X + WorkAreaOffset^[WADiPrelievo].X + 																																					(* Quota X del Cavaletto *)	
								Forming^[WorkAreaState^[WADiPrelievo].F].PackXP[NLastraDaPrelevare].X +
								Pallet^[Forming^[WorkAreaState^[WADiPrelievo].F].Pallet].OFSDE_X180;
								
			Mission^.YPick := WorkArea^[WADiPrelievo].Y + WorkAreaOffset^[WADiPrelievo].Y + 																																				(* Quota Y del Cavaletto *)						
								Forming^[WorkAreaState^[WADiPrelievo].F].PackXP[NLastraDaPrelevare].Y +
								Pallet^[Forming^[WorkAreaState^[WADiPrelievo].F].Pallet].OFSDE_Y0;
									
			Mission^.ZPick	:= WorkArea^[WADiPrelievo].Z + WorkAreaOffset^[WADiPrelievo].Z +
								Forming^[WorkAreaState^[WADiPrelievo].F].PackXP[NLastraDaPrelevare].Z +	
								Pallet^[Forming^[WorkAreaState^[WADiPrelievo].F].Pallet].OFSDE_Z0;
					
			Mission^.JPick	:= Forming^[WorkAreaState^[WADiPrelievo].F].PackXP[NLastraDaPrelevare].J +	
								Pallet^[Forming^[WorkAreaState^[WADiPrelievo].F].Pallet].OFSDE_J0;
		(*******************************************************************************************************************)						
									(* Deposito su LASTRA in cassa con rotazione piano = 90° *)
		(*******************************************************************************************************************)
		ELSE
			
			Mission^.XPick	:= WorkArea^[WADiPrelievo].X + WorkAreaOffset^[WADiPrelievo].X + 																																					(* Quota X del Cavaletto *)	
								Forming^[WorkAreaState^[WADiPrelievo].F].PackXP[NLastraDaPrelevare].X+	
								Pallet^[Forming^[WorkAreaState^[WADiPrelievo].F].Pallet].OFSDE_X90;
								
			Mission^.YPick := WorkArea^[WADiPrelievo].Y + WorkAreaOffset^[WADiPrelievo].Y + 																																				(* Quota Y del Cavaletto *)						
								Forming^[WorkAreaState^[WADiPrelievo].F].PackXP[NLastraDaPrelevare].Y + 																	(* Quota di deposito Y Ultima Lastra Depositata *)
								Pallet^[Forming^[WorkAreaState^[WADiPrelievo].F].Pallet].OFSDE_Y90;
									
			Mission^.ZPick	:= WorkArea^[WADiPrelievo].Z + WorkAreaOffset^[WADiPrelievo].Z +
								Forming^[WorkAreaState^[WADiPrelievo].F].PackXP[WADiPrelievo].Z +	
								Pallet^[Forming^[WorkAreaState^[WADiPrelievo].F].Pallet].OFSDE_Z90;
								
			Mission^.JPick	:= Forming^[WorkAreaState^[WADiPrelievo].F].PackXP[NLastraDaPrelevare].J +	
								Pallet^[Forming^[WorkAreaState^[WADiPrelievo].F].Pallet].OFSDE_J90;
		END_IF
ELSE
	Errore.Code := ErrWAM_FTC_PostazioneNONDefinita;
END_CASE

END_FUNCTION_BLOCK

// ---- POUs/TFPalletizerDataTF/TFCalcoliIngombroPinza_ConAsseK.TcPOU
(* Funzione che calcola l'ingombro della pinza nelle varie dimensioni a seconda del ciclo che la massima sta eseguendo *)
FUNCTION TFCalcoliIngombroPinza_ConAsseK : BOOL
VAR_INPUT

	Mission : POINTER TO TFMachinePalletizer_Mission;
	WorkAreaManager : POINTER TO TFWorkAreaManager;
	//
	AngoloRotazioneDestinazionePinza : LREAL; //Ango di rotazione del quale si vogliono calcolare le quote degli ingombri a destinazione  
	ModuleAX_J : POINTER TO TFModulePalletizer_AxJ_Lastre;//Modulo Asse rotazione
	//
	AngoloRotazioneDestinazionePiano : LREAL; //Angolo di rotazione del piano della pinza DESTINAZIONE => 90° = pinza parallela all'asse X
	ModuleAX_K : POINTER TO TFModulePalletizer_AxJ_Lastre;//Modulo Asse rotazione PIANO

	IngombroX_Pos : POINTER TO LREAL;//Ingombro della pinza nella Metà POSITIVA della pinza lungo X
	IngombroY_Pos : POINTER TO LREAL;//Ingombro della pinza nella Metà POSITIVA della pinza lungo Y
	
	IngombroX_Neg : POINTER TO LREAL;//Ingombro della pinza nella Metà NEGATIVA della pinza lungo X
	IngombroY_Neg : POINTER TO LREAL;//Ingombro della pinza nella Metà NEGATIVA della pinza lungo Y
	
	IngombroY_Tot : POINTER TO LREAL;//Ingombro totale In direzione Y
	
	IngombroZ_Pos : POINTER TO LREAL;//Ingombro della pinza lungo Z Positivo (sopra al fulcro)
	IngombroZ_Neg : POINTER TO LREAL;//Ingombro della pinza lungo Z Negativo (sotto al fulcro)
	
	IngombroDestinazioneX_Pos : POINTER TO LREAL;//Ingombro della pinza nella Metà POSITIVA della pinza lungo X
	IngombroDestinazioneY_Pos : POINTER TO LREAL;//Ingombro della pinza nella Metà POSITIVA della pinza lungo Y
	
	IngombroDestinazioneX_Neg : POINTER TO LREAL;//Ingombro della pinza nella Metà NEGATIVA della pinza lungo X
	IngombroDestinazioneY_Neg : POINTER TO LREAL;//Ingombro della pinza nella Metà NEGATIVA della pinza lungo Y
	
	IngombroDestinazioneZ_Pos : POINTER TO LREAL;//Ingombro della pinza lungo Z Positivo (sopra al fulcro)
	IngombroDestinazioneZ_Neg : POINTER TO LREAL;//Ingombro della pinza lungo Z Negativo (sotto al fulcro)
	
	IngombroMaxX_Pos : POINTER TO LREAL;//Ingombro MASSIMO della pinza nella Metà POSITIVA della pinza lungo X
	IngombroMaxY_Pos : POINTER TO LREAL;//Ingombro MASSIMO della pinza nella Metà POSITIVA della pinza lungo Y
	
	IngombroMaxX_Neg : POINTER TO LREAL;//Ingombro MASSIMO della pinza nella Metà NEGATIVA della pinza lungo X
	IngombroMaxY_Neg : POINTER TO LREAL;//Ingombro MASSIMO della pinza nella Metà NEGATIVA della pinza lungo Y
	
	IngombroMaxZ_Pos : POINTER TO LREAL;//Ingombro MASSIMO della pinza lungo Z Positivo (sopra al fulcro)
	IngombroMaxZ_Neg : POINTER TO LREAL;//Ingombro MASSIMO della pinza lungo Z Negativo (sotto al fulcro)

	IngombroY_Pos_0 : POINTER TO LREAL;//Ingombro della pinza nella Metà POSITIVA della pinza lungo Y
	IngombroY_Neg_180 : POINTER TO LREAL;//Ingombro della pinza nella Metà NEGATIVA della pinza lungo Y
	IngombroY_Neg_0 : POINTER TO LREAL;//Ingombro della pinza nella Metà POSITIVA della pinza lungo Y
	IngombroY_Pos_180 : POINTER TO LREAL;//Ingombro della pinza nella Metà NEGATIVA della pinza lungo Y
		
	ScostamentoVerticalePuntoCentrale : POINTER TO LREAL; //Valore che rappresenta quanto il punto centrale si è spostato rispetto allo zero orizzontale (lungo Z crescente)
END_VAR

VAR
	LunghezzaMAX 	: LREAL;//LunghezzaMAX Totale pinza
	LarghezzaMAX 	: LREAL;//Larghezza Totale pinza
	SpessoreMAX  	: LREAL;//Spessore Totale pinza	
	DimTraveVerticale : LREAL; //Dimensione Trave/Ingombro Centrale

	Diagonale			: LREAL;
	MezzaDiagonale   	: LREAL;
	Lx_MezzoAttuale : LREAL;
	Ly_MezzoAttuale : LREAL;
	Lx_MezzoDest : LREAL;
	Ly_MezzoDest : LREAL;
	Beta : LREAL;
	AngoloPerCalcoloRotPianoAttuale 	 : LREAL;
	AngoloPerCalcoloRotPianoDestinazione : LREAL;


END_VAR

(* Calcolo delle dimensioni della pinza in base al tipo di ciclo in corso *)
CASE WorkAreaManager^.State OF
	WAMANAGER_NOP,
	
	WAMANAGER_CICLO_RIPOSO_INIT:
		SpessoreMAX 	:= Dimensioni_Pinza.Spessore;
		LunghezzaMAX 	:= Dimensioni_Pinza.Lunghezza;
		LarghezzaMAX    := Dimensioni_Pinza.Larghezza;
		
	WAMANAGER_CICLO_RIPOSO_RUN:
		
		SpessoreMAX 	:= Dimensioni_Pinza.Spessore;
		LunghezzaMAX 	:= Dimensioni_Pinza.Lunghezza;
		LarghezzaMAX    := Dimensioni_Pinza.Larghezza;
															
	WAMANAGER_CICLO_PRELIEVO_FALDA_RUN:
	
		SpessoreMAX 	:= Dimensioni_Pinza.Spessore;
		LunghezzaMAX 	:= Dimensioni_Pinza.Lunghezza;
		LarghezzaMAX    := Dimensioni_Pinza.Larghezza;

	WAMANAGER_CICLO_DEPOSITO_FALDA_RUN:
		
		SpessoreMAX 	:= Dimensioni_Pinza.Spessore;
		LunghezzaMAX 	:= MAX(Dimensioni_Pinza.Lunghezza,Mission^.XDim);
		LarghezzaMAX    := MAX(Dimensioni_Pinza.Larghezza,Mission^.YDim);
										

	WAMANAGER_CICLO_PRELIEVO_LASTRA_WA_RUN:
		SpessoreMAX 	:= Dimensioni_Pinza.Spessore;
		LunghezzaMAX 	:= Dimensioni_Pinza.Lunghezza;
		LarghezzaMAX    := Dimensioni_Pinza.Larghezza;
					
	WAMANAGER_CICLO_DEPOSITO_LASTRA_SU_PAREGGIATORE_RUN:
		SpessoreMAX 	:= Dimensioni_Pinza.Spessore;
		LunghezzaMAX 	:= MAX(Dimensioni_Pinza.Lunghezza,Mission^.XDim);
		LarghezzaMAX    := MAX(Dimensioni_Pinza.Larghezza,Mission^.YDim);
					
	WAMANAGER_CICLO_PRELIEVO_LASTRA_DA_PAREGGIATORE_RUN:
	
		SpessoreMAX 	:= Dimensioni_Pinza.Spessore;
		LunghezzaMAX 	:= Dimensioni_Pinza.Lunghezza;
		LarghezzaMAX    := Dimensioni_Pinza.Larghezza;
								
	WAMANAGER_CICLO_DEPOSITO_LASTRA_WA_RUN:
	
		SpessoreMAX 	:= Dimensioni_Pinza.Spessore;
		LunghezzaMAX 	:= MAX(Dimensioni_Pinza.Lunghezza,Mission^.XDim);
		LarghezzaMAX    := MAX(Dimensioni_Pinza.Larghezza,Mission^.YDim);

	WAMANAGER_CICLO_LASTRA_PP_INIT:
		SpessoreMAX 	:= Dimensioni_Pinza.Spessore;
		LunghezzaMAX 	:= Dimensioni_Pinza.Lunghezza;
		LarghezzaMAX    := Dimensioni_Pinza.Larghezza;
						
	WAMANAGER_CICLO_PRELIEVO_LASTRA_PP_RUN:
	
		SpessoreMAX 	:= Dimensioni_Pinza.Spessore;
		LunghezzaMAX 	:= Dimensioni_Pinza.Lunghezza;
		LarghezzaMAX    := Dimensioni_Pinza.Larghezza;
						
	WAMANAGER_CICLO_DEPOSITO_LASTRA_PP_RUN:
	
		SpessoreMAX 	:= Dimensioni_Pinza.Spessore;
		LunghezzaMAX 	:= MAX(Dimensioni_Pinza.Lunghezza,Mission^.XDim);
		LarghezzaMAX    := MAX(Dimensioni_Pinza.Larghezza,Mission^.YDim);

	(* Ciclo lastra per depalettizzare da postazioni senza formature, con autoapprndimenti*)
	WAMANAGER_CICLO_PRELIEVO_LASTRA_DEPAL_RUN :
	
		SpessoreMAX 	:= Dimensioni_Pinza.Spessore;
		LunghezzaMAX 	:= Dimensioni_Pinza.Lunghezza;
		LarghezzaMAX    := Dimensioni_Pinza.Larghezza;
																				
	(* Ciclo lastra deposito su rulliera *)
	WAMANAGER_CICLO_DEPOSITO_LASTRA_DEPAL_RUN :
	
		SpessoreMAX 	:= Dimensioni_Pinza.Spessore;
		LunghezzaMAX 	:= MAX(Dimensioni_Pinza.Lunghezza,Mission^.XDim);
		LarghezzaMAX    := MAX(Dimensioni_Pinza.Larghezza,Mission^.YDim);
													
	(* Ciclo deposito FALDA su magazzino dedicato *)
	WAMANAGER_CICLO_DEPOSITO_FALDA_DEPAL_RUN :
	
		SpessoreMAX 	:= Dimensioni_Pinza.Spessore;
		LunghezzaMAX 	:= MAX(Dimensioni_Pinza.Lunghezza,Mission^.XDim);
		LarghezzaMAX    := MAX(Dimensioni_Pinza.Larghezza,Mission^.YDim);

	(* Ciclo PRELIEVO DA PANCONE *)
	WAMANAGER_CICLO_PRELIEVO_LASTRA_DA_PANCONE_RUN:
	
		SpessoreMAX 	:= Dimensioni_Pinza.Spessore;
		LunghezzaMAX 	:= Dimensioni_Pinza.Lunghezza;
		LarghezzaMAX    := Dimensioni_Pinza.Larghezza;

	(* Ciclo DEPOSITO SU PANCONE *)
	WAMANAGER_CICLO_DEPOSITO_LASTRA_SU_PANCONE_RUN:
	
		SpessoreMAX 	:= Dimensioni_Pinza.Spessore;
		LunghezzaMAX 	:= MAX(Dimensioni_Pinza.Lunghezza,Mission^.XDim);
		LarghezzaMAX    := MAX(Dimensioni_Pinza.Larghezza,Mission^.YDim);

	(* Ciclo PRELIEVO DA CANTILEVER *)
	WAMANAGER_CICLO_PRELIEVO_LASTRA_DA_CANTILEVER_RUN:
	
		SpessoreMAX 	:= Dimensioni_Pinza.Spessore;
		LunghezzaMAX 	:= Dimensioni_Pinza.Lunghezza;
		LarghezzaMAX    := Dimensioni_Pinza.Larghezza;

	(* Ciclo DEPOSITO SU CANTILEVER *)
	WAMANAGER_CICLO_DEPOSITO_LASTRA_SU_CANTILEVER_RUN:
	
		SpessoreMAX 	:= Dimensioni_Pinza.Spessore;
		LunghezzaMAX 	:= MAX(Dimensioni_Pinza.Lunghezza,Mission^.XDim);
		LarghezzaMAX    := MAX(Dimensioni_Pinza.Larghezza,Mission^.YDim);

	(* Ciclo DEPOSITO SU CANTILEVER *)
	WAMANAGER_CICLO_POSIZIONAMENTO_SEMPLICE_RUN:
	
		SpessoreMAX 	:= Dimensioni_Pinza.Spessore;
		LunghezzaMAX 	:= Dimensioni_Pinza.Lunghezza;
		LarghezzaMAX    := Dimensioni_Pinza.Larghezza;
ELSE
	SpessoreMAX 	:= Dimensioni_Pinza.Spessore;
	LunghezzaMAX 	:= MAX(Dimensioni_Pinza.Lunghezza,Mission^.XDim);
	LarghezzaMAX    := MAX(Dimensioni_Pinza.Larghezza,Mission^.YDim);
END_CASE

DimTraveVerticale := Dimensioni_Pinza.DimTraveVerticale;


Diagonale		:= SQRT(LunghezzaMAX*LunghezzaMAX+LarghezzaMAX*LarghezzaMAX);//Diagonale lastra
MezzaDiagonale	:= Diagonale/2; //Metà diagonale lastra	
Beta 			:= ATAN((LarghezzaMAX/2)/(LunghezzaMAX/2));	//Angolo dato dalla diagonale
//
AngoloPerCalcoloRotPianoAttuale := Beta + deg_to_rad(ModuleAX_K^.Ax^.AxRef^.NcToPlc.ActPos);

(* Calcolo lungo X e lungo Y i valori di ingombro a seconda di come è ruotato il piano della pinza *)
Lx_MezzoAttuale		:= ABS(MezzaDiagonale * COS(AngoloPerCalcoloRotPianoAttuale-(PI/2))); //Metà Lato "LX" parallelo all'asse X con lastra in piano
Ly_MezzoAttuale		:= ABS(MezzaDiagonale * SIN(AngoloPerCalcoloRotPianoAttuale-(PI/2))); //Metà Lato "LY" parallelo all'asse Y con lastra in piano

(* Calcolo gli ingombri in base al'angolo di rotazione della pinza *)
//IngombroX_Pos^ 	:=  LunghezzaMAX/2;
//IngombroX_Neg^ 	:=  LunghezzaMAX/2;
IngombroX_Pos^ 	:=  Lx_MezzoAttuale;// LunghezzaMAX/2;
IngombroX_Neg^ 	:=  Lx_MezzoAttuale;// LunghezzaMAX/2;


IngombroY_Neg^ 	:= MAX((Ly_MezzoAttuale * COS(deg_to_rad(-90+ModuleAX_J^.Ax^.AxRef^.NcToPlc.ActPos)) +
					SpessoreMAX * SIN(deg_to_rad(-90+ModuleAX_J^.Ax^.AxRef^.NcToPlc.ActPos))),DimTraveVerticale/2);
					
IngombroY_Pos^ 	:= ABS(MIN((-Ly_MezzoAttuale * COS(deg_to_rad(-90+ModuleAX_J^.Ax^.AxRef^.NcToPlc.ActPos)) +
					SpessoreMAX * SIN(deg_to_rad(-90+ModuleAX_J^.Ax^.AxRef^.NcToPlc.ActPos))),DimTraveVerticale/2));	

(* In base a come la pinza è ruotata inverto il positivo con il negativo in modo da avere sempre i valori corretti *)
IF AngoloRotazioneDestinazionePinza < 90 THEN	                         
	IngombroZ_Pos^	:= ABS(((Ly_MezzoAttuale) * SIN(deg_to_rad(-90+ModuleAX_J^.Ax^.AxRef^.NcToPlc.ActPos)))+
									(SpessoreMAX * COS(deg_to_rad(-90+ModuleAX_J^.Ax^.AxRef^.NcToPlc.ActPos)))-SpessoreMAX);

	IngombroZ_Neg^	:= ABS((-(Ly_MezzoAttuale) * SIN(deg_to_rad(-90+ModuleAX_J^.Ax^.AxRef^.NcToPlc.ActPos))) +
									(SpessoreMAX * COS(deg_to_rad(-90+ModuleAX_J^.Ax^.AxRef^.NcToPlc.ActPos)))-SpessoreMAX);

ELSIF  AngoloRotazioneDestinazionePinza > 90 THEN					
	IngombroZ_Pos^	:= ABS((-(Ly_MezzoAttuale) * SIN(deg_to_rad(-90+ModuleAX_J^.Ax^.AxRef^.NcToPlc.ActPos))) +
									(SpessoreMAX * COS(deg_to_rad(-90+ModuleAX_J^.Ax^.AxRef^.NcToPlc.ActPos)))-SpessoreMAX);	
	IngombroZ_Neg^	:= ABS(((Ly_MezzoAttuale) * SIN(deg_to_rad(-90+ModuleAX_J^.Ax^.AxRef^.NcToPlc.ActPos)))+
								(SpessoreMAX * COS(deg_to_rad(-90+ModuleAX_J^.Ax^.AxRef^.NcToPlc.ActPos)))-SpessoreMAX);
ELSE
	IngombroZ_Pos^	:= ABS(((Ly_MezzoAttuale) * SIN(deg_to_rad(-90+ModuleAX_J^.Ax^.AxRef^.NcToPlc.ActPos)))+
									(SpessoreMAX * COS(deg_to_rad(-90+ModuleAX_J^.Ax^.AxRef^.NcToPlc.ActPos)))-SpessoreMAX);

	IngombroZ_Neg^	:= ABS((-(Ly_MezzoAttuale) * SIN(deg_to_rad(-90+ModuleAX_J^.Ax^.AxRef^.NcToPlc.ActPos))) +
									(SpessoreMAX * COS(deg_to_rad(-90+ModuleAX_J^.Ax^.AxRef^.NcToPlc.ActPos)))-SpessoreMAX);
END_IF
IngombroY_Tot := IngombroY_Pos + IngombroY_Neg;//Ingombro TOTALE in direzione Y


(* Calcolo gli ingombri in base al'angolo di rotazione FINALE *)
AngoloPerCalcoloRotPianoDestinazione := Beta + deg_to_rad(AngoloRotazioneDestinazionePiano);

(* Calcolo lungo X e lungo Y i valori di ingombro a seconda di come è ruotato il piano della pinza *)
Lx_MezzoDest	:= ABS(MezzaDiagonale * COS(AngoloPerCalcoloRotPianoDestinazione-(PI/2))); //Metà Lato "LX" parallelo all'asse X con lastra in piano
Ly_MezzoDest	:= ABS(MezzaDiagonale * SIN(AngoloPerCalcoloRotPianoDestinazione-(PI/2))); //Metà Lato "LY" parallelo all'asse Y con lastra in piano

IngombroDestinazioneX_Pos^ 	:= Lx_MezzoDest;//  LunghezzaMAX/2;
IngombroDestinazioneX_Neg^ 	:= Ly_MezzoDest;// LunghezzaMAX/2;

IngombroDestinazioneY_Neg^ 	:= MAX((Ly_MezzoDest * COS(deg_to_rad(-90+AngoloRotazioneDestinazionePinza)) +
									SpessoreMAX * SIN(deg_to_rad(-90+AngoloRotazioneDestinazionePinza))),DimTraveVerticale/2);
					
IngombroDestinazioneY_Pos^ 	:= ABS(MIN((-Ly_MezzoDest * COS(deg_to_rad(-90+AngoloRotazioneDestinazionePinza)) +
									SpessoreMAX * SIN(deg_to_rad(-90+AngoloRotazioneDestinazionePinza))),DimTraveVerticale/2));
	
(* In base a come la pinza è ruotata inverto il positivo con il negativo in modo da avere sempre i valori corretti *)
IF AngoloRotazioneDestinazionePinza < 90 THEN	                         
	IngombroDestinazioneZ_Pos^	:= ABS(((Ly_MezzoDest) * SIN(deg_to_rad(-90+AngoloRotazioneDestinazionePinza)))+
									(SpessoreMAX * COS(deg_to_rad(-90+AngoloRotazioneDestinazionePinza)))-SpessoreMAX);

	IngombroDestinazioneZ_Neg^	:= ABS((-(Ly_MezzoDest) * SIN(deg_to_rad(-90+AngoloRotazioneDestinazionePinza))) +
									(SpessoreMAX * COS(deg_to_rad(-90+AngoloRotazioneDestinazionePinza)))-SpessoreMAX);

ELSIF  AngoloRotazioneDestinazionePinza > 90 THEN					
	IngombroDestinazioneZ_Pos^	:= ABS((-(Ly_MezzoDest) * SIN(deg_to_rad(-90+AngoloRotazioneDestinazionePinza))) +
									(SpessoreMAX * COS(deg_to_rad(-90+AngoloRotazioneDestinazionePinza)))-SpessoreMAX);	
	IngombroDestinazioneZ_Neg^	:= ABS(((Ly_MezzoDest) * SIN(deg_to_rad(-90+AngoloRotazioneDestinazionePinza)))+
								(SpessoreMAX * COS(deg_to_rad(-90+AngoloRotazioneDestinazionePinza)))-SpessoreMAX);
ELSE
	IngombroDestinazioneZ_Pos^	:= ABS(((Ly_MezzoDest) * SIN(deg_to_rad(-90+AngoloRotazioneDestinazionePinza)))+
									(SpessoreMAX * COS(deg_to_rad(-90+AngoloRotazioneDestinazionePinza)))-SpessoreMAX);

	IngombroDestinazioneZ_Neg^	:= ABS((-(Ly_MezzoDest) * SIN(deg_to_rad(-90+AngoloRotazioneDestinazionePinza))) +
									(SpessoreMAX * COS(deg_to_rad(-90+AngoloRotazioneDestinazionePinza)))-SpessoreMAX);
END_IF

(* Calcolo degli ingombri massimi nelle varie dimensioni *)
IngombroMaxX_Pos^ := MAX(IngombroX_Pos^,IngombroDestinazioneX_Pos^);//Ingombro MASSIMO della pinza nella Metà POSITIVA della pinza lungo X
IngombroMaxY_Pos^ := MAX(IngombroY_Pos^,IngombroDestinazioneY_Pos^);//Ingombro MASSIMO della pinza nella Metà POSITIVA della pinza lungo Y

IngombroMaxX_Neg^ := MAX(IngombroX_Neg^,IngombroDestinazioneX_Neg^);//Ingombro MASSIMO della pinza nella Metà NEGATIVA della pinza lungo X
IngombroMaxY_Neg^ := MAX(IngombroY_Neg^,IngombroDestinazioneY_Neg^);//Ingombro MASSIMO della pinza nella Metà NEGATIVA della pinza lungo Y

IngombroMaxZ_Pos^ := MAX(IngombroZ_Pos^,IngombroDestinazioneZ_Pos^);//Ingombro MASSIMO della pinza lungo Z Positivo (sopra al fulcro)
IngombroMaxZ_Neg^ := MAX(IngombroZ_Neg^,IngombroDestinazioneZ_Neg^);//Ingombro MASSIMO della pinza lungo Z Negativo (sotto al fulcro)


/////////////////////////////

IngombroY_Pos_0^ := ABS(MIN(SpessoreMAX * SIN(deg_to_rad(-90)),DimTraveVerticale/2));
IngombroY_Neg_180^ := ABS(MAX(SpessoreMAX * SIN(deg_to_rad(-90+180)),DimTraveVerticale/2));

IngombroY_Neg_0^ := ABS(MAX(SpessoreMAX * SIN(deg_to_rad(-90)),DimTraveVerticale/2));
IngombroY_Pos_180^ := ABS(MIN(SpessoreMAX * SIN(deg_to_rad(-90+180)),DimTraveVerticale/2));
								
ScostamentoVerticalePuntoCentrale^ := ABS(SpessoreMAX * COS(deg_to_rad(-90+AngoloRotazioneDestinazionePinza))-SpessoreMAX);
																
TFCalcoliIngombroPinza := TRUE;

END_FUNCTION

// ---- POUs/TFPalletizerDataTF/TFCalcoloTraiettoria_pacchi.TcPOU
FUNCTION_BLOCK TFCalcoloTraiettoria_pacchi
VAR_INPUT
	Traiettoria : POINTER TO TFTraiettoria;
	WorkSpace : POINTER TO TFMachinePalletizer_WorkSpace;
	WorkFootprint : POINTER TO ARRAY [1..MAXFOOTPRINT] OF TFMachinePalletizer_WorkFootprint;
	WorkPickPoint : POINTER TO ARRAY [1..MAXPICKPOINT] OF TFMachinePalletizer_WorkPickPoint;
	//WorkPickPointState : POINTER TO ARRAY [1..MAXPICKPOINT] OF TFMachinePalletizer_WorkPickPointState;

	WorkArea : POINTER TO ARRAY [1..MAXAREA] OF TFMachinePalletizer_WorkArea;
	WorkAreaState : POINTER TO ARRAY [1..MAXAREA] OF TFMachinePalletizer_WorkAreaState;
	Pallet : POINTER TO ARRAY [1..MAXPALLET] OF TFMachinePalletizer_Pallet;
	Layer : POINTER TO ARRAY [1..MAXLAYER] OF TFMachinePalletizer_Layer;
	Forming : POINTER TO ARRAY [1..MAXFORMING] OF TFMachinePalletizer_FormingForSlab;
	//ZDim : REAL;
	
	Mission : POINTER TO TFMachinePalletizer_Mission;
	
	WorkAreaManager : POINTER TO TFWorkAreaManager;
	ModuleAX_X : POINTER TO TFModulePalletizer_Ax;
	ModuleAX_Y : POINTER TO TFModulePalletizer_Ax;
	ModuleAX_Z : POINTER TO TFModulePalletizer_Ax;
	ModuleAX_J : POINTER TO TFModulePalletizer_Ax;
	ModuleAX_K : POINTER TO TFModulePalletizer_Ax;
	
END_VAR
VAR
	f : UINT;
	wa : UINT;
	P : UINT;
	a : uint;
	
	WASX : UINT;
	WADX : UINT;
	WAPARTENZA : UINT;
	WADESTINAZIONE : UINT;

	AltezzaDiIngombroArea_CCENTRALE : LREAL; //Altezza ingombro dell'Area nel corridoio CENTRALE
	AltezzaDiIngombroArea_CESTERNO : LREAL; //Altezza ingombro dell'Area nel corridoio ESTERNO
	AltezzaDiIngombroArea_CINTERNO : LREAL; //Altezza ingombro dell'Area nel corridoio INTERNO
	
	
	
	
	AltezzaDiIngombroOstacoli : LREAL;
	AltezzaDiIngombroPuntiPrelievo : LREAL;
	AssegnaQuote : BOOL;
	OffsetSicurezzaConPacco : REAL;
	AltezzaPinzaDaTastatoreAFlangiaMotore : REAL; // Altezza della pinza dal tastatore al bordo superiore della flangia di supporto motore asse K
	AltezzaDaPavimentoAPiastraSupportoColonnaCentrale : REAL;
	LarghezzaPiastraSupportoColonnaCentrale : REAL;
	Quota_X_CentroColonnaCentrale : REAL;
END_VAR

(* Ingombri colonna centrale *)
(*AltezzaPinzaDaTastatoreAFlangiaMotore := 270;
AltezzaDaPavimentoAPiastraSupportoColonnaCentrale := 2070;
LarghezzaPiastraSupportoColonnaCentrale := 500;
Quota_X_CentroColonnaCentrale := 7545;*)

CASE WorkAreaManager^.State OF
	WAMANAGER_NOP,
	
	WAMANAGER_CICLO_RIPOSO_INIT,
		
	WAMANAGER_CICLO_RIPOSO_RUN:
		IF Mission^.State = MISSION_STATE_NOP THEN
			QuotaFuoriIngombro_Z_AVUOTO_CCENTRALE := 0;
			(* Valuto gli ostacoli *)	
			FOR f:=1 TO MAXFOOTPRINT DO	
				IF QuotaFuoriIngombro_Z_AVUOTO_CCENTRALE <= WorkFootPrint^[f].Z + WorkFootPrint^[f].ZDim + TCPParameter.Z + OffsetSicurezza.Avuoto THEN
					QuotaFuoriIngombro_Z_AVUOTO_CCENTRALE := WorkFootPrint^[f].Z + WorkFootPrint^[f].ZDim + TCPParameter.Z + OffsetSicurezza.Avuoto;
				END_IF
			END_FOR
			(* Valuto le aree *)
			FOR a:=1 TO MAXAREA DO
				AltezzaDiIngombroArea_CCENTRALE := 0;
				IF WorkAreaState^[a].H > WorkAreaState^[a].HPL THEN
					AltezzaDiIngombroArea_CCENTRALE := WorkAreaState^[a].H;
				ELSE
					AltezzaDiIngombroArea_CCENTRALE := WorkAreaState^[a].HPL;
				END_IF
				(* Se ho la postazione falde e/o catasta vuoti con riscontri fissi metto la quota fissa di altezza della postazione all'altezza massima*)
				IF WorkArea^[a].Typology = TYPOLOGY_LAYER THEN
					AltezzaDiIngombroArea_CCENTRALE := ALTEZZA_CATASTA_FALDE;
				ELSIF  WorkArea^[a].Typology <> TYPOLOGY_STACK AND CATASTA_VUOTI_CON_RISCONTRI_FISSI THEN
					AltezzaDiIngombroArea_CCENTRALE := ALTEZZA_CATASTA_VUOTI;
				END_IF
				
				IF QuotaFuoriIngombro_Z_AVUOTO_CCENTRALE <= AltezzaDiIngombroArea_CCENTRALE + TCPParameter.Z + OffsetSicurezza.Avuoto  THEN
					QuotaFuoriIngombro_Z_AVUOTO_CCENTRALE := AltezzaDiIngombroArea_CCENTRALE + TCPParameter.Z + OffsetSicurezza.Avuoto;
				END_IF
			END_FOR
			
			
			/////////////////////////////////////////////////////////////!!!!!!!!!!!!!!!!!!!!!!!!!!!!!!!!//////////////////////////////
			IF TFDirezioneAssePositiva(Posizione_Attuale:=ModuleAX_X^.Ax^.Status.ActPosition,Posizione_Finale:=Mission^.XPick) THEN	// Direzione Positiva 
				(*TFCalcolaNumeroPostazioneDXSX(PosizioneAttuale:=ModuleAX_X^.Ax^.Status.ActPosition,
												WorkArea:=WorkArea,
												DirezioneAsseX_Positiva:=TRUE,
												NPostazioneDX=>WADX,
												NPostazioneSX=>WASX,
												PostazionePartenza=>WAPARTENZA);*)
												
				IF WorkArea^[wa].Typology <> TYPOLOGY_EXTERNAL_DEPPREL THEN
					FOR wa := WAPARTENZA TO NumPostazioneDiPareggiatura DO
						AltezzaDiIngombroArea_CCENTRALE := 0;
						CASE WorkArea^[wa].Typology OF
							TYPOLOGY_PALLET:
								CASE Forming^[WorkAreaState^[wa].F].Pallet.Tipologia OF
										
									PALLET_STANDARD:
										IF WorkAreaState^[wa].H > WorkAreaState^[wa].HPL THEN
											AltezzaDiIngombroArea_CCENTRALE := WorkAreaState^[wa].H;
										ELSE
											AltezzaDiIngombroArea_CCENTRALE := WorkAreaState^[wa].HPL;
										END_IF
										IF WorkArea^[wa].Z > AltezzaDiIngombroArea_CCENTRALE THEN
											AltezzaDiIngombroArea_CCENTRALE := WorkArea^[wa].Z;	
										END_IF
									
									CASSA_STANDARD:
										IF Forming^[WorkAreaState^[wa].F].Pallet.HMAX > WorkAreaState^[wa].H THEN
											AltezzaDiIngombroArea_CCENTRALE := Forming^[WorkAreaState^[wa].F].Pallet.HMAX;
										ELSE
											AltezzaDiIngombroArea_CCENTRALE := WorkAreaState^[wa].H;
										END_IF
										IF WorkArea^[wa].Z > AltezzaDiIngombroArea_CCENTRALE THEN
											AltezzaDiIngombroArea_CCENTRALE := WorkArea^[wa].Z;	
										END_IF
										
									CAVALLETTO:
										IF Forming^[WorkAreaState^[wa].F].Pallet.HMAX > WorkAreaState^[wa].H THEN
											AltezzaDiIngombroArea_CCENTRALE := Forming^[WorkAreaState^[wa].F].Pallet.HMAX;
										ELSE
											AltezzaDiIngombroArea_CCENTRALE := WorkAreaState^[wa].H;
										END_IF
										IF WorkArea^[wa].Z > AltezzaDiIngombroArea_CCENTRALE THEN
											AltezzaDiIngombroArea_CCENTRALE := WorkArea^[wa].Z;	
										END_IF
										
									ELSE
										AltezzaDiIngombroArea_CCENTRALE := 1700;//Fisso l'altezza ad una quota di default
								END_CASE
											
							TYPOLOGY_LAYER:
								IF WorkAreaState^[wa].H > WorkAreaState^[wa].HPL THEN
									AltezzaDiIngombroArea_CCENTRALE := WorkAreaState^[wa].H;
								ELSE
									AltezzaDiIngombroArea_CCENTRALE := WorkAreaState^[wa].HPL;
								END_IF
								IF WorkArea^[wa].Z > AltezzaDiIngombroArea_CCENTRALE THEN
									AltezzaDiIngombroArea_CCENTRALE := WorkArea^[wa].Z;	
								END_IF
							
							TYPOLOGY_EXTERNAL_DEPPREL:
								AltezzaDiIngombroArea_CCENTRALE := AltezzaDiIngombroArea_CCENTRALE;
								
							ELSE
								AltezzaDiIngombroArea_CCENTRALE := 1700;//Fisso l'altezza ad una quota di default
						
						END_CASE					
																
						IF QuotaFuoriIngombro_Z_AVUOTO_CCENTRALE <= AltezzaDiIngombroArea_CCENTRALE + TCPParameter.Z + OffsetSicurezza.Avuoto  THEN
							QuotaFuoriIngombro_Z_AVUOTO_CCENTRALE := AltezzaDiIngombroArea_CCENTRALE + TCPParameter.Z + OffsetSicurezza.Avuoto;
						END_IF
					END_FOR	
				END_IF	
			ELSE
				(*TFCalcolaNumeroPostazioneDXSX(PosizioneAttuale	:= ModuleAX_X^.Ax^.Status.ActPosition,
												WorkArea		:= WorkArea,
												DirezioneAsseX_Positiva:=FALSE,
												NPostazioneDX	=> WADX,
												NPostazioneSX	=> WASX,
												PostazionePartenza=>WAPARTENZA);*)
						
				FOR wa := WAPARTENZA TO NPOSTAZIONE_DOPODELPUNTODIPREL BY -1 DO
					AltezzaDiIngombroArea_CCENTRALE := 0;
					IF WorkAreaState^[wa].H > WorkAreaState^[wa].HPL THEN
						AltezzaDiIngombroArea_CCENTRALE := WorkAreaState^[wa].H;
					ELSE
						AltezzaDiIngombroArea_CCENTRALE := WorkAreaState^[wa].HPL;
					END_IF
					IF QuotaFuoriIngombro_Z_AVUOTO_CCENTRALE <= AltezzaDiIngombroArea_CCENTRALE + TCPParameter.Z + OffsetSicurezza.Avuoto  THEN
						QuotaFuoriIngombro_Z_AVUOTO_CCENTRALE := AltezzaDiIngombroArea_CCENTRALE + TCPParameter.Z + OffsetSicurezza.Avuoto;
					END_IF
				END_FOR			
					(* Valuto I Pick-Point *)
					(*FOR P:=1 TO MAXPICKPOINT DO
						AltezzaDiIngombroPuntiPrelievo := 0;
						IF  WorkPickPoint^[P].Zh + WorkPickPointState^[P].ZDim >= WorkPickPointDimension[P].Zdim THEN // Se Altezza orrizzontale Ribaltino + Zpacco >= Ingombro Verticale Ribaltino
							AltezzaDiIngombroPuntiPrelievo := WorkPickPoint^[P].Zh + WorkPickPointState^[P].ZDim;
						END_IF
						IF WorkPickPoint^[P].Zv + WorkPickPointState^[P].ZTilter + WorkPickPointState^[P].YDim >= WorkPickPointDimension[P].Zdim THEN // Se Altezza Vertivale Ribaltino + Quota Fermo + Ypacco >= Ingombro Verticale Ribaltino
							AltezzaDiIngombroPuntiPrelievo := WorkPickPoint^[P].Zv + WorkPickPointState^[P].ZTilter + WorkPickPointState^[P].YDim;
						END_IF
						IF WorkPickPointDimension[P].Zdim >= AltezzaDiIngombroPuntiPrelievo THEN //Se Ingombro Verticale Ribaltino >= Dell'ingombro valutato sopra
							AltezzaDiIngombroPuntiPrelievo := WorkPickPointDimension[P].Zdim;
						END_IF
						IF WAPARTENZA = NPOSTAZIONE_PRIMADELPUNTODIPREL THEN //Se sono nella posizione 7 valuto l'altezza del ribaltino "REALE", con o senza pacco
							IF QuotaAnticipoDinamicaZ_VersoRiposo <= AltezzaDiIngombroPuntiPrelievo + TCPParameter.Z + OffsetSicurezza.Avuoto THEN //Se Quota fuori ingombro <= dell' ingombro del punto di prelievo
								QuotaAnticipoDinamicaZ_VersoRiposo := AltezzaDiIngombroPuntiPrelievo + TCPParameter.Z + OffsetSicurezza.Avuoto;
							END_IF
						ELSE		//Se non sono nella WA 7, do una quota fittizzia, inferiore all'altezza del ribaltino "reale"
							IF QuotaAnticipoDinamicaZ_VersoRiposo <= AltezzaDiIngombroPuntiPrelievo + TCPParameter.Z + OffsetSicurezzaAnticipoMovimenti.OffsetSicurezzaAnticipo_Z - 300 THEN
								QuotaAnticipoDinamicaZ_VersoRiposo := AltezzaDiIngombroPuntiPrelievo + WorkPickPointState^[P].YDim + TCPParameter.Z + OffsetSicurezzaAnticipoMovimenti.OffsetSicurezzaAnticipo_Z - 300;
							END_IF
						END_IF
					END_FOR*)
				//END_IF
				IF ModuleAX_Z^.Ax^.Status.ActPosition >= QuotaAnticipoDinamicaZ_VersoRiposo THEN
					QuotaAnticipoDinamicaZ_Raggiunta := TRUE;
				ELSE
					QuotaAnticipoDinamicaZ_Raggiunta := FALSE;
				END_IF
			
			
			
			END_IF
				(* Valuto I Pick-Point *)
				CASE TIPOLOGIA_FUNZIONAMENTO_MACCHINA OF
					
					FUNZIONAMENTO_PICKING:
						AltezzaDiIngombroPuntiPrelievo := 0;
															
				ELSE;
					(*FOR P:=1 TO MAXPICKPOINT DO
						AltezzaDiIngombroPuntiPrelievo := 0;
						IF  WorkPickPointDimension^[P].Zdim + WorkPickPointState^[P].Element.Z >= WorkPickPointDimension^[P].Zdim THEN // Se Altezza + Zpacco >= Ingombro Verticale 
							AltezzaDiIngombroPuntiPrelievo := WorkPickPoint^[P].Z + WorkPickPointState^[P].Element.Z;
						END_IF
						IF WorkPickPointDimension^[P].Zdim >= AltezzaDiIngombroPuntiPrelievo THEN //Se Ingombro Verticale >= Dell'ingombro valutato sopra
							AltezzaDiIngombroPuntiPrelievo := WorkPickPointDimension^[P].Zdim;
						END_IF
						//Se non sono nella WA 7, do una quota fittizzia, inferiore all'altezza del ribaltino "reale"
						IF QuotaAnticipoDinamicaZ_VersoRiposo <= AltezzaDiIngombroPuntiPrelievo + TCPParameter.Z + OffsetSicurezzaAnticipoMovimenti.OffsetSicurezzaAnticipo_Z - 300 THEN
							QuotaAnticipoDinamicaZ_VersoRiposo := AltezzaDiIngombroPuntiPrelievo + WorkPickPointState^[P].Element.YDim + TCPParameter.Z + OffsetSicurezzaAnticipoMovimenti.OffsetSicurezzaAnticipo_Z - 300;
						END_IF
					END_FOR		*)	
				END_CASE
			
			
			
			
			
		END_IF //riferito all'IF dello stato della missione	
												
	WAMANAGER_CICLO_RIPOSO_END,
	(*		
	WAMANAGER_CICLO_PALL_INIT,
	
